// @TEST-ASSERT
AssertTrue(Condition := equal, Message := 'Did not convert LREAL to DINT correctly');
AssertTrue(Condition := converted, Message := 'Did not report LREAL to DINT conversion was successful');

TEST_FINISHED();
END_METHOD

METHOD PUBLIC Check_LREAL_TO_DT_Min
VAR
	value : LREAL := DatatypeLimits.MIN_VALUE_OF_LREAL_WHICH_CAN_BE_HELD_IN_A_DT;
	actual : DT;
	converted : BOOL;
	equal : BOOL;
END_VAR
TEST('Check_LREAL_TO_DT_Min');

// @TEST-RUN
converted := TryConvert_LREAL_TO_Destination(value, actual);
equal := actual = LREAL_TO_DT(value);

// @TEST-ASSERT
AssertTrue(Condition := equal, Message := 'Did not convert LREAL to DT correctly');
AssertTrue(Condition := converted, Message := 'Did not report LREAL to DT conversion was successful');

TEST_FINISHED();
END_METHOD

METHOD PUBLIC Check_LREAL_TO_DT_TooHigh
VAR
	value : LREAL := DatatypeLimits.LREAL_MAX_VALUE;
	actual : DT;
	converted : BOOL;
END_VAR
TEST('Check_LREAL_TO_DT_TooHigh');

// @TEST-RUN
converted := TryConvert_LREAL_TO_Destination(value, actual);

// @TEST-ASSERT
AssertFalse(Condition := converted, Message := 'Did not report LREAL to DT conversion was prevented');

TEST_FINISHED();
END_METHOD

METHOD PUBLIC Check_LREAL_TO_DT_TooLow
VAR
	value : LREAL := DatatypeLimits.LREAL_MIN_VALUE;
	actual : DT;
	converted : BOOL;
END_VAR
TEST('Check_LREAL_TO_DT_TooLow');

// @TEST-RUN
converted := TryConvert_LREAL_TO_Destination(value, actual);

// @TEST-ASSERT
AssertFalse(Condition := converted, Message := 'Did not report LREAL to DT conversion was prevented');

TEST_FINISHED();
END_METHOD

METHOD PUBLIC Check_LREAL_TO_DT_Max
VAR
	value : LREAL := DatatypeLimits.MAX_VALUE_OF_LREAL_WHICH_CAN_BE_HELD_IN_A_DT;
	actual : DT;
	converted : BOOL;
	equal : BOOL;
END_VAR
TEST('Check_LREAL_TO_DT_Max');

// @TEST-RUN
converted := TryConvert_LREAL_TO_Destination(value, actual);
equal := actual = LREAL_TO_DT(value);

// @TEST-ASSERT
AssertTrue(Condition := equal, Message := 'Did not convert LREAL to DT correctly');
AssertTrue(Condition := converted, Message := 'Did not report LREAL to DT conversion was successful');

TEST_FINISHED();
END_METHOD

METHOD PUBLIC Check_LREAL_TO_DWORD_Min
VAR
	value : LREAL := DatatypeLimits.MIN_VALUE_OF_LREAL_WHICH_CAN_BE_HELD_IN_A_DWORD;
	actual : DWORD;
	converted : BOOL;
	equal : BOOL;
END_VAR
TEST('Check_LREAL_TO_DWORD_Min');

// @TEST-RUN
converted := TryConvert_LREAL_TO_Destination(value, actual);
equal := actual = LREAL_TO_DWORD(value);

// @TEST-ASSERT
AssertTrue(Condition := equal, Message := 'Did not convert LREAL to DWORD correctly');
AssertTrue(Condition := converted, Message := 'Did not report LREAL to DWORD conversion was successful');

TEST_FINISHED();
END_METHOD

METHOD PUBLIC Check_LREAL_TO_DWORD_TooHigh
VAR
	value : LREAL := DatatypeLimits.LREAL_MAX_VALUE;
	actual : DWORD;
	converted : BOOL;
END_VAR
TEST('Check_LREAL_TO_DWORD_TooHigh');

// @TEST-RUN
converted := TryConvert_LREAL_TO_Destination(value, actual);

// @TEST-ASSERT
AssertFalse(Condition := converted, Message := 'Did not report LREAL to DWORD conversion was prevented');

TEST_FINISHED();
END_METHOD

METHOD PUBLIC Check_LREAL_TO_DWORD_TooLow
VAR
	value : LREAL := DatatypeLimits.LREAL_MIN_VALUE;
	actual : DWORD;
	converted : BOOL;
END_VAR
TEST('Check_LREAL_TO_DWORD_TooLow');

// @TEST-RUN
converted := TryConvert_LREAL_TO_Destination(value, actual);

// @TEST-ASSERT
AssertFalse(Condition := converted, Message := 'Did not report LREAL to DWORD conversion was prevented');

TEST_FINISHED();
END_METHOD

METHOD PUBLIC Check_LREAL_TO_DWORD_Max
VAR
	value : LREAL := DatatypeLimits.MAX_VALUE_OF_LREAL_WHICH_CAN_BE_HELD_IN_A_DWORD;
	actual : DWORD;
	converted : BOOL;
	equal : BOOL;
END_VAR
TEST('Check_LREAL_TO_DWORD_Max');

// @TEST-RUN
converted := TryConvert_LREAL_TO_Destination(value, actual);
equal := actual = LREAL_TO_DWORD(value);

// @TEST-ASSERT
AssertTrue(Condition := equal, Message := 'Did not convert LREAL to DWORD correctly');
AssertTrue(Condition := converted, Message := 'Did not report LREAL to DWORD conversion was successful');

TEST_FINISHED();
END_METHOD

METHOD PUBLIC Check_LREAL_TO_INT_Min
VAR
	value : LREAL := DatatypeLimits.MIN_VALUE_OF_LREAL_WHICH_CAN_BE_HELD_IN_A_INT;
	actual : INT;
	converted : BOOL;
	equal : BOOL;
END_VAR
TEST('Check_LREAL_TO_INT_Min');

// @TEST-RUN
converted := TryConvert_LREAL_TO_Destination(value, actual);
equal := actual = LREAL_TO_INT(value);

// @TEST-ASSERT
AssertTrue(Condition := equal, Message := 'Did not convert LREAL to INT correctly');
AssertTrue(Condition := converted, Message := 'Did not report LREAL to INT conversion was successful');

TEST_FINISHED();
END_METHOD

METHOD PUBLIC Check_LREAL_TO_INT_TooHigh
VAR
	value : LREAL := DatatypeLimits.LREAL_MAX_VALUE;
	actual : INT;
	converted : BOOL;
END_VAR
TEST('Check_LREAL_TO_INT_TooHigh');

// @TEST-RUN
converted := TryConvert_LREAL_TO_Destination(value, actual);

// @TEST-ASSERT
AssertFalse(Condition := converted, Message := 'Did not report LREAL to INT conversion was prevented');

TEST_FINISHED();
END_METHOD

METHOD PUBLIC Check_LREAL_TO_INT_TooLow
VAR
	value : LREAL := DatatypeLimits.LREAL_MIN_VALUE;
	actual : INT;
	converted : BOOL;
END_VAR
TEST('Check_LREAL_TO_INT_TooLow');

// @TEST-RUN
converted := TryConvert_LREAL_TO_Destination(value, actual);

// @TEST-ASSERT
AssertFalse(Condition := converted, Message := 'Did not report LREAL to INT conversion was prevented');

TEST_FINISHED();
END_METHOD

METHOD PUBLIC Check_LREAL_TO_INT_Max
VAR
	value : LREAL := DatatypeLimits.MAX_VALUE_OF_LREAL_WHICH_CAN_BE_HELD_IN_A_INT;
	actual : INT;
	converted : BOOL;
	equal : BOOL;
END_VAR
TEST('Check_LREAL_TO_INT_Max');

// @TEST-RUN
converted := TryConvert_LREAL_TO_Destination(value, actual);
equal := actual = LREAL_TO_INT(value);

// @TEST-ASSERT
AssertTrue(Condition := equal, Message := 'Did not convert LREAL to INT correctly');
AssertTrue(Condition := converted, Message := 'Did not report LREAL to INT conversion was successful');

TEST_FINISHED();
END_METHOD

METHOD PUBLIC Check_LREAL_TO_LINT_Min
VAR
	value : LREAL := DatatypeLimits.MIN_VALUE_OF_LREAL_WHICH_CAN_BE_HELD_IN_A_LINT;
	actual : LINT;
	converted : BOOL;
	equal : BOOL;
END_VAR
TEST('Check_LREAL_TO_LINT_Min');

// @TEST-RUN
converted := TryConvert_LREAL_TO_Destination(value, actual);
equal := actual = LREAL_TO_LINT(value);

// @TEST-ASSERT
AssertTrue(Condition := equal, Message := 'Did not convert LREAL to LINT correctly');
AssertTrue(Condition := converted, Message := 'Did not report LREAL to LINT conversion was successful');

TEST_FINISHED();
END_METHOD

METHOD PUBLIC Check_LREAL_TO_LINT_TooHigh
VAR
	value : LREAL := DatatypeLimits.LREAL_MAX_VALUE;
	actual : LINT;
	converted : BOOL;
END_VAR
TEST('Check_LREAL_TO_LINT_TooHigh');

// @TEST-RUN
converted := TryConvert_LREAL_TO_Destination(value, actual);

// @TEST-ASSERT
AssertFalse(Condition := converted, Message := 'Did not report LREAL to LINT conversion was prevented');

TEST_FINISHED();
END_METHOD

METHOD PUBLIC Check_LREAL_TO_LINT_TooLow
VAR
	value : LREAL := DatatypeLimits.LREAL_MIN_VALUE;
	actual : LINT;
	converted : BOOL;
END_VAR
TEST('Check_LREAL_TO_LINT_TooLow');

// @TEST-RUN
converted := TryConvert_LREAL_TO_Destination(value, actual);

// @TEST-ASSERT
AssertFalse(Condition := converted, Message := 'Did not report LREAL to LINT conversion was prevented');

TEST_FINISHED();
END_METHOD

METHOD PUBLIC Check_LREAL_TO_LINT_Max
VAR
	value : LREAL := DatatypeLimits.MAX_VALUE_OF_LREAL_WHICH_CAN_BE_HELD_IN_A_LINT;
	actual : LINT;
	converted : BOOL;
	equal : BOOL;
END_VAR
TEST('Check_LREAL_TO_LINT_Max');

// @TEST-RUN
converted := TryConvert_LREAL_TO_Destination(value, actual);
equal := actual = LREAL_TO_LINT(value);

// @TEST-ASSERT
AssertTrue(Condition := equal, Message := 'Did not convert LREAL to LINT correctly');
AssertTrue(Condition := converted, Message := 'Did not report LREAL to LINT conversion was successful');

TEST_FINISHED();
END_METHOD

METHOD PUBLIC Check_LREAL_TO_LREAL_Min
VAR
	value : LREAL := DatatypeLimits.LREAL_MIN_VALUE;
	actual : LREAL;
	converted : BOOL;
	equal : BOOL;
END_VAR
TEST('Check_LREAL_TO_LREAL_Min');

// @TEST-RUN
converted := TryConvert_LREAL_TO_Destination(value, actual);
equal := actual = value;

// @TEST-ASSERT
AssertTrue(Condition := equal, Message := 'Did not convert LREAL to LREAL correctly');
AssertTrue(Condition := converted, Message := 'Did not report LREAL to LREAL conversion was successful');

TEST_FINISHED();
END_METHOD

METHOD PUBLIC Check_LREAL_TO_LREAL_Max
VAR
	value : LREAL := DatatypeLimits.LREAL_MAX_VALUE;
	actual : LREAL;
	converted : BOOL;
	equal : BOOL;
END_VAR
TEST('Check_LREAL_TO_LREAL_Max');

// @TEST-RUN
converted := TryConvert_LREAL_TO_Destination(value, actual);
equal := actual = value;

// @TEST-ASSERT
AssertTrue(Condition := equal, Message := 'Did not convert LREAL to LREAL correctly');
AssertTrue(Condition := converted, Message := 'Did not report LREAL to LREAL conversion was successful');

TEST_FINISHED();
END_METHOD

METHOD PUBLIC Check_LREAL_TO_LWORD_Min
VAR
	value : LREAL := DatatypeLimits.MIN_VALUE_OF_LREAL_WHICH_CAN_BE_HELD_IN_A_LWORD;
	actual : LWORD;
	converted : BOOL;
	equal : BOOL;
END_VAR
TEST('Check_LREAL_TO_LWORD_Min');

// @TEST-RUN
converted := TryConvert_LREAL_TO_Destination(value, actual);
equal := actual = LREAL_TO_LWORD(value);

// @TEST-ASSERT
AssertTrue(Condition := equal, Message := 'Did not convert LREAL to LWORD correctly');
AssertTrue(Condition := converted, Message := 'Did not report LREAL to LWORD conversion was successful');

TEST_FINISHED();
END_METHOD

METHOD PUBLIC Check_LREAL_TO_LWORD_TooHigh
VAR
	value : LREAL := DatatypeLimits.LREAL_MAX_VALUE;
	actual : LWORD;
	converted : BOOL;
END_VAR
TEST('Check_LREAL_TO_LWORD_TooHigh');

// @TEST-RUN
converted := TryConvert_LREAL_TO_Destination(value, actual);

// @TEST-ASSERT
AssertFalse(Condition := converted, Message := 'Did not report LREAL to LWORD conversion was prevented');

TEST_FINISHED();
END_METHOD

METHOD PUBLIC Check_LREAL_TO_LWORD_TooLow
VAR
	value : LREAL := DatatypeLimits.LREAL_MIN_VALUE;
	actual : LWORD;
	converted : BOOL;
END_VAR
TEST('Check_LREAL_TO_LWORD_TooLow');

// @TEST-RUN
converted := TryConvert_LREAL_TO_Destination(value, actual);

// @TEST-ASSERT
AssertFalse(Condition := converted, Message := 'Did not report LREAL to LWORD conversion was prevented');

TEST_FINISHED();
END_METHOD

METHOD PUBLIC Check_LREAL_TO_LWORD_Max
VAR
	value : LREAL := DatatypeLimits.MAX_VALUE_OF_LREAL_WHICH_CAN_BE_HELD_IN_A_LWORD;
	actual : LWORD;
	converted : BOOL;
	equal : BOOL;
END_VAR
TEST('Check_LREAL_TO_LWORD_Max');

// @TEST-RUN
converted := TryConvert_LREAL_TO_Destination(value, actual);
equal := actual = LREAL_TO_LWORD(value);

// @TEST-ASSERT
AssertTrue(Condition := equal, Message := 'Did not convert LREAL to LWORD correctly');
AssertTrue(Condition := converted, Message := 'Did not report LREAL to LWORD conversion was successful');

TEST_FINISHED();
END_METHOD

METHOD PUBLIC Check_LREAL_TO_REAL_Min
VAR
	value : LREAL := DatatypeLimits.MIN_VALUE_OF_LREAL_WHICH_CAN_BE_HELD_IN_A_REAL;
	actual : REAL;
	converted : BOOL;
	equal : BOOL;
END_VAR
TEST('Check_LREAL_TO_REAL_Min');

// @TEST-RUN
converted := TryConvert_LREAL_TO_Destination(value, actual);
equal := actual = LREAL_TO_REAL(value);

// @TEST-ASSERT
AssertTrue(Condition := equal, Message := 'Did not convert LREAL to REAL correctly');
AssertTrue(Condition := converted, Message := 'Did not report LREAL to REAL conversion was successful');

TEST_FINISHED();
END_METHOD

METHOD PUBLIC Check_LREAL_TO_REAL_TooHigh
VAR
	value : LREAL := DatatypeLimits.LREAL_MAX_VALUE;
	actual : REAL;
	converted : BOOL;
END_VAR
TEST('Check_LREAL_TO_REAL_TooHigh');

// @TEST-RUN
converted := TryConvert_LREAL_TO_Destination(value, actual);

// @TEST-ASSERT
AssertFalse(Condition := converted, Message := 'Did not report LREAL to REAL conversion was prevented');

TEST_FINISHED();
END_METHOD

METHOD PUBLIC Check_LREAL_TO_REAL_TooLow
VAR
	value : LREAL := DatatypeLimits.LREAL_MIN_VALUE;
	actual : REAL;
	converted : BOOL;
END_VAR
TEST('Check_LREAL_TO_REAL_TooLow');

// @TEST-RUN
converted := TryConvert_LREAL_TO_Destination(value, actual);

// @TEST-ASSERT
AssertFalse(Condition := converted, Message := 'Did not report LREAL to REAL conversion was prevented');

TEST_FINISHED();
END_METHOD

METHOD PUBLIC Check_LREAL_TO_REAL_Max
VAR
	value : LREAL := DatatypeLimits.MAX_VALUE_OF_LREAL_WHICH_CAN_BE_HELD_IN_A_REAL;
	actual : REAL;
	converted : BOOL;
	equal : BOOL;
END_VAR
TEST('Check_LREAL_TO_REAL_Max');

// @TEST-RUN
converted := TryConvert_LREAL_TO_Destination(value, actual);
equal := actual = LREAL_TO_REAL(value);

// @TEST-ASSERT
AssertTrue(Condition := equal, Message := 'Did not convert LREAL to REAL correctly');
AssertTrue(Condition := converted, Message := 'Did not report LREAL to REAL conversion was successful');

TEST_FINISHED();
END_METHOD

METHOD PUBLIC Check_LREAL_TO_SINT_Min
VAR
	value : LREAL := DatatypeLimits.MIN_VALUE_OF_LREAL_WHICH_CAN_BE_HELD_IN_A_SINT;
	actual : SINT;
	converted : BOOL;
	equal : BOOL;
END_VAR
TEST('Check_LREAL_TO_SINT_Min');

// @TEST-RUN
converted := TryConvert_LREAL_TO_Destination(value, actual);
equal := actual = LREAL_TO_SINT(value);

// @TEST-ASSERT
AssertTrue(Condition := equal, Message := 'Did not convert LREAL to SINT correctly');
AssertTrue(Condition := converted, Message := 'Did not report LREAL to SINT conversion was successful');

TEST_FINISHED();
END_METHOD

METHOD PUBLIC Check_LREAL_TO_SINT_TooHigh
VAR
	value : LREAL := DatatypeLimits.LREAL_MAX_VALUE;
	actual : SINT;
	converted : BOOL;
END_VAR
TEST('Check_LREAL_TO_SINT_TooHigh');

// @TEST-RUN
converted := TryConvert_LREAL_TO_Destination(value, actual);

// @TEST-ASSERT
AssertFalse(Condition := converted, Message := 'Did not report LREAL to SINT conversion was prevented');

TEST_FINISHED();
END_METHOD

METHOD PUBLIC Check_LREAL_TO_SINT_TooLow
VAR
	value : LREAL := DatatypeLimits.LREAL_MIN_VALUE;
	actual : SINT;
	converted : BOOL;
END_VAR
TEST('Check_LREAL_TO_SINT_TooLow');

// @TEST-RUN
converted := TryConvert_LREAL_TO_Destination(value, actual);

// @TEST-ASSERT
AssertFalse(Condition := converted, Message := 'Did not report LREAL to SINT conversion was prevented');

TEST_FINISHED();
END_METHOD

METHOD PUBLIC Check_LREAL_TO_SINT_Max
VAR
	value : LREAL := DatatypeLimits.MAX_VALUE_OF_LREAL_WHICH_CAN_BE_HELD_IN_A_SINT;
	actual : SINT;
	converted : BOOL;
	equal : BOOL;
END_VAR
TEST('Check_LREAL_TO_SINT_Max');

// @TEST-RUN
converted := TryConvert_LREAL_TO_Destination(value, actual);
equal := actual = LREAL_TO_SINT(value);

// @TEST-ASSERT
AssertTrue(Condition := equal, Message := 'Did not convert LREAL to SINT correctly');
AssertTrue(Condition := converted, Message := 'Did not report LREAL to SINT conversion was successful');

TEST_FINISHED();
END_METHOD

METHOD PUBLIC Check_LREAL_TO_STRING_Min
VAR
	value : LREAL := DatatypeLimits.MIN_VALUE_OF_LREAL_WHICH_CAN_BE_HELD_IN_A_STRING;
	actual : STRING;
	converted : BOOL;
	equal : BOOL;
END_VAR
TEST('Check_LREAL_TO_STRING_Min');

// @TEST-RUN
converted := TryConvert_LREAL_TO_Destination(value, actual);
equal := actual = LREAL_TO_STRING(value);

// @TEST-ASSERT
AssertTrue(Condition := equal, Message := 'Did not convert LREAL to STRING correctly');
AssertTrue(Condition := converted, Message := 'Did not report LREAL to STRING conversion was successful');

TEST_FINISHED();
END_METHOD

METHOD PUBLIC Check_LREAL_TO_STRING_TooHigh
VAR
	value : LREAL := DatatypeLimits.LREAL_MAX_VALUE;
	actual : STRING;
	converted : BOOL;
END_VAR
TEST('Check_LREAL_TO_STRING_TooHigh');

// @TEST-RUN
converted := TryConvert_LREAL_TO_Destination(value, actual);

// @TEST-ASSERT
AssertFalse(Condition := converted, Message := 'Did not report LREAL to STRING conversion was prevented');

TEST_FINISHED();
END_METHOD

METHOD PUBLIC Check_LREAL_TO_STRING_TooLow
VAR
	value : LREAL := DatatypeLimits.LREAL_MIN_VALUE;
	actual : STRING;
	converted : BOOL;
END_VAR
TEST('Check_LREAL_TO_STRING_TooLow');

// @TEST-RUN
converted := TryConvert_LREAL_TO_Destination(value, actual);

// @TEST-ASSERT
AssertFalse(Condition := converted, Message := 'Did not report LREAL to STRING conversion was prevented');

TEST_FINISHED();
END_METHOD

METHOD PUBLIC Check_LREAL_TO_STRING_Max
VAR
	value : LREAL := DatatypeLimits.MAX_VALUE_OF_LREAL_WHICH_CAN_BE_HELD_IN_A_STRING;
	actual : STRING;
	converted : BOOL;
	equal : BOOL;
END_VAR
TEST('Check_LREAL_TO_STRING_Max');

// @TEST-RUN
converted := TryConvert_LREAL_TO_Destination(value, actual);
equal := actual = LREAL_TO_STRING(value);

// @TEST-ASSERT
AssertTrue(Condition := equal, Message := 'Did not convert LREAL to STRING correctly');
AssertTrue(Condition := converted, Message := 'Did not report LREAL to STRING conversion was successful');

TEST_FINISHED();
END_METHOD

METHOD PUBLIC Check_LREAL_TO_TIME_Min
VAR
	value : LREAL := DatatypeLimits.MIN_VALUE_OF_LREAL_WHICH_CAN_BE_HELD_IN_A_TIME;
	actual : TIME;
	converted : BOOL;
	equal : BOOL;
END_VAR
TEST('Check_LREAL_TO_TIME_Min');

// @TEST-RUN
converted := TryConvert_LREAL_TO_Destination(value, actual);
equal := actual = LREAL_TO_TIME(value);

// @TEST-ASSERT
AssertTrue(Condition := equal, Message := 'Did not convert LREAL to TIME correctly');
AssertTrue(Condition := converted, Message := 'Did not report LREAL to TIME conversion was successful');

TEST_FINISHED();
END_METHOD

METHOD PUBLIC Check_LREAL_TO_TIME_TooHigh
VAR
	value : LREAL := DatatypeLimits.LREAL_MAX_VALUE;
	actual : TIME;
	converted : BOOL;
END_VAR
TEST('Check_LREAL_TO_TIME_TooHigh');

// @TEST-RUN
converted := TryConvert_LREAL_TO_Destination(value, actual);

// @TEST-ASSERT
AssertFalse(Condition := converted, Message := 'Did not report LREAL to TIME conversion was prevented');

TEST_FINISHED();
END_METHOD

METHOD PUBLIC Check_LREAL_TO_TIME_TooLow
VAR
	value : LREAL := DatatypeLimits.LREAL_MIN_VALUE;
	actual : TIME;
	converted : BOOL;
END_VAR
TEST('Check_LREAL_TO_TIME_TooLow');

// @TEST-RUN
converted := TryConvert_LREAL_TO_Destination(value, actual);

// @TEST-ASSERT
AssertFalse(Condition := converted, Message := 'Did not report LREAL to TIME conversion was prevented');

TEST_FINISHED();
END_METHOD

METHOD PUBLIC Check_LREAL_TO_TIME_Max
VAR
	value : LREAL := DatatypeLimits.MAX_VALUE_OF_LREAL_WHICH_CAN_BE_HELD_IN_A_TIME;
	actual : TIME;
	converted : BOOL;
	equal : BOOL;
END_VAR
TEST('Check_LREAL_TO_TIME_Max');

// @TEST-RUN
converted := TryConvert_LREAL_TO_Destination(value, actual);
equal := actual = LREAL_TO_TIME(value);

// @TEST-ASSERT
AssertTrue(Condition := equal, Message := 'Did not convert LREAL to TIME correctly');
AssertTrue(Condition := converted, Message := 'Did not report LREAL to TIME conversion was successful');

TEST_FINISHED();
END_METHOD

METHOD PUBLIC Check_LREAL_TO_TOD_Min
VAR
	value : LREAL := DatatypeLimits.MIN_VALUE_OF_LREAL_WHICH_CAN_BE_HELD_IN_A_TOD;
	actual : TOD;
	converted : BOOL;
	equal : BOOL;
END_VAR
TEST('Check_LREAL_TO_TOD_Min');

// @TEST-RUN
converted := TryConvert_LREAL_TO_Destination(value, actual);
equal := actual = LREAL_TO_TOD(value);

// @TEST-ASSERT
AssertTrue(Condition := equal, Message := 'Did not convert LREAL to TOD correctly');
AssertTrue(Condition := converted, Message := 'Did not report LREAL to TOD conversion was successful');

TEST_FINISHED();
END_METHOD

METHOD PUBLIC Check_LREAL_TO_TOD_TooHigh
VAR
	value : LREAL := DatatypeLimits.LREAL_MAX_VALUE;
	actual : TOD;
	converted : BOOL;
END_VAR
TEST('Check_LREAL_TO_TOD_TooHigh');

// @TEST-RUN
converted := TryConvert_LREAL_TO_Destination(value, actual);

// @TEST-ASSERT
AssertFalse(Condition := converted, Message := 'Did not report LREAL to TOD conversion was prevented');

TEST_FINISHED();
END_METHOD

METHOD PUBLIC Check_LREAL_TO_TOD_TooLow
VAR
	value : LREAL := DatatypeLimits.LREAL_MIN_VALUE;
	actual : TOD;
	converted : BOOL;
END_VAR
TEST('Check_LREAL_TO_TOD_TooLow');

// @TEST-RUN
converted := TryConvert_LREAL_TO_Destination(value, actual);

// @TEST-ASSERT
AssertFalse(Condition := converted, Message := 'Did not report LREAL to TOD conversion was prevented');

TEST_FINISHED();
END_METHOD

METHOD PUBLIC Check_LREAL_TO_TOD_Max
VAR
	value : LREAL := DatatypeLimits.MAX_VALUE_OF_LREAL_WHICH_CAN_BE_HELD_IN_A_TOD;
	actual : TOD;
	converted : BOOL;
	equal : BOOL;
END_VAR
TEST('Check_LREAL_TO_TOD_Max');

// @TEST-RUN
converted := TryConvert_LREAL_TO_Destination(value, actual);
equal := actual = LREAL_TO_TOD(value);

// @TEST-ASSERT
AssertTrue(Condition := equal, Message := 'Did not convert LREAL to TOD correctly');
AssertTrue(Condition := converted, Message := 'Did not report LREAL to TOD conversion was successful');

TEST_FINISHED();
END_METHOD

METHOD PUBLIC Check_LREAL_TO_UDINT_Min
VAR
	value : LREAL := DatatypeLimits.MIN_VALUE_OF_LREAL_WHICH_CAN_BE_HELD_IN_A_UDINT;
	actual : UDINT;
	converted : BOOL;
	equal : BOOL;
END_VAR
TEST('Check_LREAL_TO_UDINT_Min');

// @TEST-RUN
converted := TryConvert_LREAL_TO_Destination(value, actual);
equal := actual = LREAL_TO_UDINT(value);

// @TEST-ASSERT
AssertTrue(Condition := equal, Message := 'Did not convert LREAL to UDINT correctly');
AssertTrue(Condition := converted, Message := 'Did not report LREAL to UDINT conversion was successful');

TEST_FINISHED();
END_METHOD

METHOD PUBLIC Check_LREAL_TO_UDINT_TooHigh
VAR
	value : LREAL := DatatypeLimits.LREAL_MAX_VALUE;
	actual : UDINT;
	converted : BOOL;
END_VAR
TEST('Check_LREAL_TO_UDINT_TooHigh');

// @TEST-RUN
converted := TryConvert_LREAL_TO_Destination(value, actual);

// @TEST-ASSERT
AssertFalse(Condition := converted, Message := 'Did not report LREAL to UDINT conversion was prevented');

TEST_FINISHED();
END_METHOD

METHOD PUBLIC Check_LREAL_TO_UDINT_TooLow
VAR
	value : LREAL := DatatypeLimits.LREAL_MIN_VALUE;
	actual : UDINT;
	converted : BOOL;
END_VAR
TEST('Check_LREAL_TO_UDINT_TooLow');

// @TEST-RUN
converted := TryConvert_LREAL_TO_Destination(value, actual);

// @TEST-ASSERT
AssertFalse(Condition := converted, Message := 'Did not report LREAL to UDINT conversion was prevented');

TEST_FINISHED();
END_METHOD

METHOD PUBLIC Check_LREAL_TO_UDINT_Max
VAR
	value : LREAL := DatatypeLimits.MAX_VALUE_OF_LREAL_WHICH_CAN_BE_HELD_IN_A_UDINT;
	actual : UDINT;
	converted : BOOL;
	equal : BOOL;
END_VAR
TEST('Check_LREAL_TO_UDINT_Max');

// @TEST-RUN
converted := TryConvert_LREAL_TO_Destination(value, actual);
equal := actual = LREAL_TO_UDINT(value);

// @TEST-ASSERT
AssertTrue(Condition := equal, Message := 'Did not convert LREAL to UDINT correctly');
AssertTrue(Condition := converted, Message := 'Did not report LREAL to UDINT conversion was successful');

TEST_FINISHED();
END_METHOD

METHOD PUBLIC Check_LREAL_TO_UINT_Min
VAR
	value : LREAL := DatatypeLimits.MIN_VALUE_OF_LREAL_WHICH_CAN_BE_HELD_IN_A_UINT;
	actual : UINT;
	converted : BOOL;
	equal : BOOL;
END_VAR
TEST('Check_LREAL_TO_UINT_Min');

// @TEST-RUN
converted := TryConvert_LREAL_TO_Destination(value, actual);
equal := actual = LREAL_TO_UINT(value);

// @TEST-ASSERT
AssertTrue(Condition := equal, Message := 'Did not convert LREAL to UINT correctly');
AssertTrue(Condition := converted, Message := 'Did not report LREAL to UINT conversion was successful');

TEST_FINISHED();
END_METHOD

METHOD PUBLIC Check_LREAL_TO_UINT_TooHigh
VAR
	value : LREAL := DatatypeLimits.LREAL_MAX_VALUE;
	actual : UINT;
	converted : BOOL;
END_VAR
TEST('Check_LREAL_TO_UINT_TooHigh');

// @TEST-RUN
converted := TryConvert_LREAL_TO_Destination(value, actual);

// @TEST-ASSERT
AssertFalse(Condition := converted, Message := 'Did not report LREAL to UINT conversion was prevented');

TEST_FINISHED();
END_METHOD

METHOD PUBLIC Check_LREAL_TO_UINT_TooLow
VAR
	value : LREAL := DatatypeLimits.LREAL_MIN_VALUE;
	actual : UINT;
	converted : BOOL;
END_VAR
TEST('Check_LREAL_TO_UINT_TooLow');

// @TEST-RUN
converted := TryConvert_LREAL_TO_Destination(value, actual);

// @TEST-ASSERT
AssertFalse(Condition := converted, Message := 'Did not report LREAL to UINT conversion was prevented');

TEST_FINISHED();
END_METHOD

METHOD PUBLIC Check_LREAL_TO_UINT_Max
VAR
	value : LREAL := DatatypeLimits.MAX_VALUE_OF_LREAL_WHICH_CAN_BE_HELD_IN_A_UINT;
	actual : UINT;
	converted : BOOL;
	equal : BOOL;
END_VAR
TEST('Check_LREAL_TO_UINT_Max');

// @TEST-RUN
converted := TryConvert_LREAL_TO_Destination(value, actual);
equal := actual = LREAL_TO_UINT(value);

// @TEST-ASSERT
AssertTrue(Condition := equal, Message := 'Did not convert LREAL to UINT correctly');
AssertTrue(Condition := converted, Message := 'Did not report LREAL to UINT conversion was successful');

TEST_FINISHED();
END_METHOD

METHOD PUBLIC Check_LREAL_TO_ULINT_Min
VAR
	value : LREAL := DatatypeLimits.MIN_VALUE_OF_LREAL_WHICH_CAN_BE_HELD_IN_A_ULINT;
	actual : ULINT;
	converted : BOOL;
	equal : BOOL;
END_VAR
TEST('Check_LREAL_TO_ULINT_Min');

// @TEST-RUN
converted := TryConvert_LREAL_TO_Destination(value, actual);
equal := actual = LREAL_TO_ULINT(value);

// @TEST-ASSERT
AssertTrue(Condition := equal, Message := 'Did not convert LREAL to ULINT correctly');
AssertTrue(Condition := converted, Message := 'Did not report LREAL to ULINT conversion was successful');

TEST_FINISHED();
END_METHOD

METHOD PUBLIC Check_LREAL_TO_ULINT_TooHigh
VAR
	value : LREAL := DatatypeLimits.LREAL_MAX_VALUE;
	actual : ULINT;
	converted : BOOL;
END_VAR
TEST('Check_LREAL_TO_ULINT_TooHigh');

// @TEST-RUN
converted := TryConvert_LREAL_TO_Destination(value, actual);

// @TEST-ASSERT
AssertFalse(Condition := converted, Message := 'Did not report LREAL to ULINT conversion was prevented');

TEST_FINISHED();
END_METHOD

METHOD PUBLIC Check_LREAL_TO_ULINT_TooLow
VAR
	value : LREAL := DatatypeLimits.LREAL_MIN_VALUE;
	actual : ULINT;
	converted : BOOL;
END_VAR
TEST('Check_LREAL_TO_ULINT_TooLow');

// @TEST-RUN
converted := TryConvert_LREAL_TO_Destination(value, actual);

// @TEST-ASSERT
AssertFalse(Condition := converted, Message := 'Did not report LREAL to ULINT conversion was prevented');

TEST_FINISHED();
END_METHOD

METHOD PUBLIC Check_LREAL_TO_ULINT_Max
VAR
	value : LREAL := DatatypeLimits.MAX_VALUE_OF_LREAL_WHICH_CAN_BE_HELD_IN_A_ULINT;
	actual : ULINT;
	converted : BOOL;
	equal : BOOL;
END_VAR
TEST('Check_LREAL_TO_ULINT_Max');

// @TEST-RUN
converted := TryConvert_LREAL_TO_Destination(value, actual);
equal := actual = LREAL_TO_ULINT(value);

// @TEST-ASSERT
AssertTrue(Condition := equal, Message := 'Did not convert LREAL to ULINT correctly');
AssertTrue(Condition := converted, Message := 'Did not report LREAL to ULINT conversion was successful');

TEST_FINISHED();
END_METHOD

METHOD PUBLIC Check_LREAL_TO_USINT_Min
VAR
	value : LREAL := DatatypeLimits.MIN_VALUE_OF_LREAL_WHICH_CAN_BE_HELD_IN_A_USINT;
	actual : USINT;
	converted : BOOL;
	equal : BOOL;
END_VAR
TEST('Check_LREAL_TO_USINT_Min');

// @TEST-RUN
converted := TryConvert_LREAL_TO_Destination(value, actual);
equal := actual = LREAL_TO_USINT(value);

// @TEST-ASSERT
AssertTrue(Condition := equal, Message := 'Did not convert LREAL to USINT correctly');
AssertTrue(Condition := converted, Message := 'Did not report LREAL to USINT conversion was successful');

TEST_FINISHED();
END_METHOD

METHOD PUBLIC Check_LREAL_TO_USINT_TooHigh
VAR
	value : LREAL := DatatypeLimits.LREAL_MAX_VALUE;
	actual : USINT;
	converted : BOOL;
END_VAR
TEST('Check_LREAL_TO_USINT_TooHigh');

// @TEST-RUN
converted := TryConvert_LREAL_TO_Destination(value, actual);

// @TEST-ASSERT
AssertFalse(Condition := converted, Message := 'Did not report LREAL to USINT conversion was prevented');

TEST_FINISHED();
END_METHOD

METHOD PUBLIC Check_LREAL_TO_USINT_TooLow
VAR
	value : LREAL := DatatypeLimits.LREAL_MIN_VALUE;
	actual : USINT;
	converted : BOOL;
END_VAR
TEST('Check_LREAL_TO_USINT_TooLow');

// @TEST-RUN
converted := TryConvert_LREAL_TO_Destination(value, actual);

// @TEST-ASSERT
AssertFalse(Condition := converted, Message := 'Did not report LREAL to USINT conversion was prevented');

TEST_FINISHED();
END_METHOD

METHOD PUBLIC Check_LREAL_TO_USINT_Max
VAR
	value : LREAL := DatatypeLimits.MAX_VALUE_OF_LREAL_WHICH_CAN_BE_HELD_IN_A_USINT;
	actual : USINT;
	converted : BOOL;
	equal : BOOL;
END_VAR
TEST('Check_LREAL_TO_USINT_Max');

// @TEST-RUN
converted := TryConvert_LREAL_TO_Destination(value, actual);
equal := actual = LREAL_TO_USINT(value);

// @TEST-ASSERT
AssertTrue(Condition := equal, Message := 'Did not convert LREAL to USINT correctly');
AssertTrue(Condition := converted, Message := 'Did not report LREAL to USINT conversion was successful');

TEST_FINISHED();
END_METHOD

METHOD PUBLIC Check_LREAL_TO_WORD_Min
VAR
	value : LREAL := DatatypeLimits.MIN_VALUE_OF_LREAL_WHICH_CAN_BE_HELD_IN_A_WORD;
	actual : WORD;
	converted : BOOL;
	equal : BOOL;
END_VAR
TEST('Check_LREAL_TO_WORD_Min');

// @TEST-RUN
converted := TryConvert_LREAL_TO_Destination(value, actual);
equal := actual = LREAL_TO_WORD(value);

// @TEST-ASSERT
AssertTrue(Condition := equal, Message := 'Did not convert LREAL to WORD correctly');
AssertTrue(Condition := converted, Message := 'Did not report LREAL to WORD conversion was successful');

TEST_FINISHED();
END_METHOD

METHOD PUBLIC Check_LREAL_TO_WORD_TooHigh
VAR
	value : LREAL := DatatypeLimits.LREAL_MAX_VALUE;
	actual : WORD;
	converted : BOOL;
END_VAR
TEST('Check_LREAL_TO_WORD_TooHigh');

// @TEST-RUN
converted := TryConvert_LREAL_TO_Destination(value, actual);

// @TEST-ASSERT
AssertFalse(Condition := converted, Message := 'Did not report LREAL to WORD conversion was prevented');

TEST_FINISHED();
END_METHOD

METHOD PUBLIC Check_LREAL_TO_WORD_TooLow
VAR
	value : LREAL := DatatypeLimits.LREAL_MIN_VALUE;
	actual : WORD;
	converted : BOOL;
END_VAR
TEST('Check_LREAL_TO_WORD_TooLow');

// @TEST-RUN
converted := TryConvert_LREAL_TO_Destination(value, actual);

// @TEST-ASSERT
AssertFalse(Condition := converted, Message := 'Did not report LREAL to WORD conversion was prevented');

TEST_FINISHED();
END_METHOD

METHOD PUBLIC Check_LREAL_TO_WORD_Max
VAR
	value : LREAL := DatatypeLimits.MAX_VALUE_OF_LREAL_WHICH_CAN_BE_HELD_IN_A_WORD;
	actual : WORD;
	converted : BOOL;
	equal : BOOL;
END_VAR
TEST('Check_LREAL_TO_WORD_Max');

// @TEST-RUN
converted := TryConvert_LREAL_TO_Destination(value, actual);
equal := actual = LREAL_TO_WORD(value);

// @TEST-ASSERT
AssertTrue(Condition := equal, Message := 'Did not convert LREAL to WORD correctly');
AssertTrue(Condition := converted, Message := 'Did not report LREAL to WORD conversion was successful');

TEST_FINISHED();
END_METHOD

END_FUNCTION_BLOCK

// ---- Tests/TIME_TO_TestSuite.TcPOU
FUNCTION_BLOCK PUBLIC TIME_TO_TestSuite EXTENDS TcUnit.FB_TestSuite
VAR
END_VAR

Check_TIME_TO_BOOL_Max();
Check_TIME_TO_BOOL_Min();
Check_TIME_TO_BYTE_Max();
Check_TIME_TO_BYTE_Min();
Check_TIME_TO_BYTE_TooHigh();
Check_TIME_TO_WORD_Max();
Check_TIME_TO_WORD_Min();
Check_TIME_TO_WORD_TooHigh();
Check_TIME_TO_DWORD_Max();
Check_TIME_TO_DWORD_Min();
Check_TIME_TO_LWORD_Max();
Check_TIME_TO_LWORD_Min();
Check_TIME_TO_SINT_Max();
Check_TIME_TO_SINT_Min();
Check_TIME_TO_SINT_TooHigh();
Check_TIME_TO_INT_Max();
Check_TIME_TO_INT_Min();
Check_TIME_TO_INT_TooHigh();
Check_TIME_TO_DINT_Max();
Check_TIME_TO_DINT_Min();
Check_TIME_TO_DINT_TooHigh();
Check_TIME_TO_LINT_Max();
Check_TIME_TO_LINT_Min();
Check_TIME_TO_USINT_Max();
Check_TIME_TO_USINT_Min();
Check_TIME_TO_USINT_TooHigh();
Check_TIME_TO_UINT_Max();
Check_TIME_TO_UINT_Min();
Check_TIME_TO_UINT_TooHigh();
Check_TIME_TO_UDINT_Max();
Check_TIME_TO_UDINT_Min();
Check_TIME_TO_ULINT_Max();
Check_TIME_TO_ULINT_Min();
Check_TIME_TO_REAL_Max();
Check_TIME_TO_REAL_Min();
Check_TIME_TO_LREAL_Max();
Check_TIME_TO_LREAL_Min();
Check_TIME_TO_TIME_Max();
Check_TIME_TO_TIME_Min();
Check_TIME_TO_TOD_Max();
Check_TIME_TO_TOD_Min();
Check_TIME_TO_TOD_TooHigh();
Check_TIME_TO_DATE_Max();
Check_TIME_TO_DATE_Min();
Check_TIME_TO_DT_Max();
Check_TIME_TO_DT_Min();
Check_TIME_TO_STRING_Max();
Check_TIME_TO_STRING_Min();

METHOD PUBLIC Check_TIME_TO_BOOL_Min
VAR
	value : TIME := DatatypeLimits.TIME_MIN_VALUE;
	actual : BOOL;
	converted : BOOL;
	equal : BOOL;
END_VAR
TEST('Check_TIME_TO_BOOL_Min');

// @TEST-RUN
converted := TryConvert_TIME_TO_Destination(value, actual);
equal := actual = TIME_TO_BOOL(value);

// @TEST-ASSERT
AssertTrue(Condition := equal, Message := 'Did not convert TIME to BOOL correctly');
AssertTrue(Condition := converted, Message := 'Did not report TIME to BOOL conversion was successful');

TEST_FINISHED();
END_METHOD

METHOD PUBLIC Check_TIME_TO_BOOL_Max
VAR
	value : TIME := DatatypeLimits.TIME_MAX_VALUE;
	actual : BOOL;
	converted : BOOL;
	equal : BOOL;
END_VAR
TEST('Check_TIME_TO_BOOL_Max');

// @TEST-RUN
converted := TryConvert_TIME_TO_Destination(value, actual);
equal := actual = TIME_TO_BOOL(value);

// @TEST-ASSERT
AssertTrue(Condition := equal, Message := 'Did not convert TIME to BOOL correctly');
AssertTrue(Condition := converted, Message := 'Did not report TIME to BOOL conversion was successful');

TEST_FINISHED();
END_METHOD

METHOD PUBLIC Check_TIME_TO_BYTE_Min
VAR
	value : TIME := DatatypeLimits.TIME_MIN_VALUE;
	actual : BYTE;
	converted : BOOL;
	equal : BOOL;
END_VAR
TEST('Check_TIME_TO_BYTE_Min');

// @TEST-RUN
converted := TryConvert_TIME_TO_Destination(value, actual);
equal := actual = TIME_TO_BYTE(value);

// @TEST-ASSERT
AssertTrue(Condition := equal, Message := 'Did not convert TIME to BYTE correctly');
AssertTrue(Condition := converted, Message := 'Did not report TIME to BYTE conversion was successful');

TEST_FINISHED();
END_METHOD

METHOD PUBLIC Check_TIME_TO_BYTE_TooHigh
VAR
	value : TIME := DatatypeLimits.TIME_MAX_VALUE;
	actual : BYTE;
	converted : BOOL;
END_VAR
TEST('Check_TIME_TO_BYTE_TooHigh');

// @TEST-RUN
converted := TryConvert_TIME_TO_Destination(value, actual);

// @TEST-ASSERT
AssertFalse(Condition := converted, Message := 'Did not report TIME to BYTE conversion was prevented');

TEST_FINISHED();
END_METHOD

METHOD PUBLIC Check_TIME_TO_BYTE_Max
VAR
	value : TIME := DatatypeLimits.MAX_VALUE_OF_TIME_WHICH_CAN_BE_HELD_IN_A_BYTE;
	actual : BYTE;
	converted : BOOL;
	equal : BOOL;
END_VAR
TEST('Check_TIME_TO_BYTE_Max');

// @TEST-RUN
converted := TryConvert_TIME_TO_Destination(value, actual);
equal := actual = TIME_TO_BYTE(value);

// @TEST-ASSERT
AssertTrue(Condition := equal, Message := 'Did not convert TIME to BYTE correctly');
AssertTrue(Condition := converted, Message := 'Did not report TIME to BYTE conversion was successful');

TEST_FINISHED();
END_METHOD

METHOD PUBLIC Check_TIME_TO_DATE_Min
VAR
	value : TIME := DatatypeLimits.TIME_MIN_VALUE;
	actual : DATE;
	converted : BOOL;
	equal : BOOL;
END_VAR
TEST('Check_TIME_TO_DATE_Min');

// @TEST-RUN
converted := TryConvert_TIME_TO_Destination(value, actual);
equal := actual = TIME_TO_DATE(value);

// @TEST-ASSERT
AssertTrue(Condition := equal, Message := 'Did not convert TIME to DATE correctly');
AssertTrue(Condition := converted, Message := 'Did not report TIME to DATE conversion was successful');

TEST_FINISHED();
END_METHOD

METHOD PUBLIC Check_TIME_TO_DATE_Max
VAR
	value : TIME := DatatypeLimits.TIME_MAX_VALUE;
	actual : DATE;
	converted : BOOL;
	equal : BOOL;
END_VAR
TEST('Check_TIME_TO_DATE_Max');

// @TEST-RUN
converted := TryConvert_TIME_TO_Destination(value, actual);
equal := actual = TIME_TO_DATE(value);

// @TEST-ASSERT
AssertTrue(Condition := equal, Message := 'Did not convert TIME to DATE correctly');
AssertTrue(Condition := converted, Message := 'Did not report TIME to DATE conversion was successful');

TEST_FINISHED();
END_METHOD

METHOD PUBLIC Check_TIME_TO_DINT_Min
VAR
	value : TIME := DatatypeLimits.TIME_MIN_VALUE;
	actual : DINT;
	converted : BOOL;
	equal : BOOL;
END_VAR
TEST('Check_TIME_TO_DINT_Min');

// @TEST-RUN
converted := TryConvert_TIME_TO_Destination(value, actual);
equal := actual = TIME_TO_DINT(value);

// @TEST-ASSERT
AssertTrue(Condition := equal, Message := 'Did not convert TIME to DINT correctly');
AssertTrue(Condition := converted, Message := 'Did not report TIME to DINT conversion was successful');

TEST_FINISHED();
END_METHOD

METHOD PUBLIC Check_TIME_TO_DINT_TooHigh
VAR
	value : TIME := DatatypeLimits.TIME_MAX_VALUE;
	actual : DINT;
	converted : BOOL;
END_VAR
TEST('Check_TIME_TO_DINT_TooHigh');

// @TEST-RUN
converted := TryConvert_TIME_TO_Destination(value, actual);

// @TEST-ASSERT
AssertFalse(Condition := converted, Message := 'Did not report TIME to DINT conversion was prevented');

TEST_FINISHED();
END_METHOD

METHOD PUBLIC Check_TIME_TO_DINT_Max
VAR
	value : TIME := DatatypeLimits.MAX_VALUE_OF_TIME_WHICH_CAN_BE_HELD_IN_A_DINT;
	actual : DINT;
	converted : BOOL;
	equal : BOOL;
END_VAR
TEST('Check_TIME_TO_DINT_Max');

// @TEST-RUN
converted := TryConvert_TIME_TO_Destination(value, actual);
equal := actual = TIME_TO_DINT(value);

// @TEST-ASSERT
AssertTrue(Condition := equal, Message := 'Did not convert TIME to DINT correctly');
AssertTrue(Condition := converted, Message := 'Did not report TIME to DINT conversion was successful');

TEST_FINISHED();
END_METHOD

METHOD PUBLIC Check_TIME_TO_DT_Min
VAR
	value : TIME := DatatypeLimits.TIME_MIN_VALUE;
	actual : DT;
	converted : BOOL;
	equal : BOOL;
END_VAR
TEST('Check_TIME_TO_DT_Min');

// @TEST-RUN
converted := TryConvert_TIME_TO_Destination(value, actual);
equal := actual = TIME_TO_DT(value);

// @TEST-ASSERT
AssertTrue(Condition := equal, Message := 'Did not convert TIME to DT correctly');
AssertTrue(Condition := converted, Message := 'Did not report TIME to DT conversion was successful');

TEST_FINISHED();
END_METHOD

METHOD PUBLIC Check_TIME_TO_DT_Max
VAR
	value : TIME := DatatypeLimits.TIME_MAX_VALUE;
	actual : DT;
	converted : BOOL;
	equal : BOOL;
END_VAR
TEST('Check_TIME_TO_DT_Max');

// @TEST-RUN
converted := TryConvert_TIME_TO_Destination(value, actual);
equal := actual = TIME_TO_DT(value);

// @TEST-ASSERT
AssertTrue(Condition := equal, Message := 'Did not convert TIME to DT correctly');
AssertTrue(Condition := converted, Message := 'Did not report TIME to DT conversion was successful');

TEST_FINISHED();
END_METHOD

METHOD PUBLIC Check_TIME_TO_DWORD_Min
VAR
	value : TIME := DatatypeLimits.TIME_MIN_VALUE;
	actual : DWORD;
	converted : BOOL;
	equal : BOOL;
END_VAR
TEST('Check_TIME_TO_DWORD_Min');

// @TEST-RUN
converted := TryConvert_TIME_TO_Destination(value, actual);
equal := actual = TIME_TO_DWORD(value);

// @TEST-ASSERT
AssertTrue(Condition := equal, Message := 'Did not convert TIME to DWORD correctly');
AssertTrue(Condition := converted, Message := 'Did not report TIME to DWORD conversion was successful');

TEST_FINISHED();
END_METHOD

METHOD PUBLIC Check_TIME_TO_DWORD_Max
VAR
	value : TIME := DatatypeLimits.TIME_MAX_VALUE;
	actual : DWORD;
	converted : BOOL;
	equal : BOOL;
END_VAR
TEST('Check_TIME_TO_DWORD_Max');

// @TEST-RUN
converted := TryConvert_TIME_TO_Destination(value, actual);
equal := actual = TIME_TO_DWORD(value);

// @TEST-ASSERT
AssertTrue(Condition := equal, Message := 'Did not convert TIME to DWORD correctly');
AssertTrue(Condition := converted, Message := 'Did not report TIME to DWORD conversion was successful');

TEST_FINISHED();
END_METHOD

METHOD PUBLIC Check_TIME_TO_INT_Min
VAR
	value : TIME := DatatypeLimits.TIME_MIN_VALUE;
	actual : INT;
	converted : BOOL;
	equal : BOOL;
END_VAR
TEST('Check_TIME_TO_INT_Min');

// @TEST-RUN
converted := TryConvert_TIME_TO_Destination(value, actual);
equal := actual = TIME_TO_INT(value);

// @TEST-ASSERT
AssertTrue(Condition := equal, Message := 'Did not convert TIME to INT correctly');
AssertTrue(Condition := converted, Message := 'Did not report TIME to INT conversion was successful');

TEST_FINISHED();
END_METHOD

METHOD PUBLIC Check_TIME_TO_INT_TooHigh
VAR
	value : TIME := DatatypeLimits.TIME_MAX_VALUE;
	actual : INT;
	converted : BOOL;
END_VAR
TEST('Check_TIME_TO_INT_TooHigh');

// @TEST-RUN
converted := TryConvert_TIME_TO_Destination(value, actual);

// @TEST-ASSERT
AssertFalse(Condition := converted, Message := 'Did not report TIME to INT conversion was prevented');

TEST_FINISHED();
END_METHOD

METHOD PUBLIC Check_TIME_TO_INT_Max
VAR
	value : TIME := DatatypeLimits.MAX_VALUE_OF_TIME_WHICH_CAN_BE_HELD_IN_A_INT;
	actual : INT;
	converted : BOOL;
	equal : BOOL;
END_VAR
TEST('Check_TIME_TO_INT_Max');

// @TEST-RUN
converted := TryConvert_TIME_TO_Destination(value, actual);
equal := actual = TIME_TO_INT(value);

// @TEST-ASSERT
AssertTrue(Condition := equal, Message := 'Did not convert TIME to INT correctly');
AssertTrue(Condition := converted, Message := 'Did not report TIME to INT conversion was successful');

TEST_FINISHED();
END_METHOD

METHOD PUBLIC Check_TIME_TO_LINT_Min
VAR
	value : TIME := DatatypeLimits.TIME_MIN_VALUE;
	actual : LINT;
	converted : BOOL;
	equal : BOOL;
END_VAR
TEST('Check_TIME_TO_LINT_Min');

// @TEST-RUN
converted := TryConvert_TIME_TO_Destination(value, actual);
equal := actual = TIME_TO_LINT(value);

// @TEST-ASSERT
AssertTrue(Condition := equal, Message := 'Did not convert TIME to LINT correctly');
AssertTrue(Condition := converted, Message := 'Did not report TIME to LINT conversion was successful');

TEST_FINISHED();
END_METHOD

METHOD PUBLIC Check_TIME_TO_LINT_Max
VAR
	value : TIME := DatatypeLimits.TIME_MAX_VALUE;
	actual : LINT;
	converted : BOOL;
	equal : BOOL;
END_VAR
TEST('Check_TIME_TO_LINT_Max');

// @TEST-RUN
converted := TryConvert_TIME_TO_Destination(value, actual);
equal := actual = TIME_TO_LINT(value);

// @TEST-ASSERT
AssertTrue(Condition := equal, Message := 'Did not convert TIME to LINT correctly');
AssertTrue(Condition := converted, Message := 'Did not report TIME to LINT conversion was successful');

TEST_FINISHED();
END_METHOD

METHOD PUBLIC Check_TIME_TO_LREAL_Min
VAR
	value : TIME := DatatypeLimits.TIME_MIN_VALUE;
	actual : LREAL;
	converted : BOOL;
	equal : BOOL;
END_VAR
TEST('Check_TIME_TO_LREAL_Min');

// @TEST-RUN
converted := TryConvert_TIME_TO_Destination(value, actual);
equal := actual = TIME_TO_LREAL(value);

// @TEST-ASSERT
AssertTrue(Condition := equal, Message := 'Did not convert TIME to LREAL correctly');
AssertTrue(Condition := converted, Message := 'Did not report TIME to LREAL conversion was successful');

TEST_FINISHED();
END_METHOD

METHOD PUBLIC Check_TIME_TO_LREAL_Max
VAR
	value : TIME := DatatypeLimits.TIME_MAX_VALUE;
	actual : LREAL;
	converted : BOOL;
	equal : BOOL;
END_VAR
TEST('Check_TIME_TO_LREAL_Max');

// @TEST-RUN
converted := TryConvert_TIME_TO_Destination(value, actual);
equal := actual = TIME_TO_LREAL(value);

// @TEST-ASSERT
AssertTrue(Condition := equal, Message := 'Did not convert TIME to LREAL correctly');
AssertTrue(Condition := converted, Message := 'Did not report TIME to LREAL conversion was successful');

TEST_FINISHED();
END_METHOD

METHOD PUBLIC Check_TIME_TO_LWORD_Min
VAR
	value : TIME := DatatypeLimits.TIME_MIN_VALUE;
	actual : LWORD;
	converted : BOOL;
	equal : BOOL;
END_VAR
TEST('Check_TIME_TO_LWORD_Min');

// @TEST-RUN
converted := TryConvert_TIME_TO_Destination(value, actual);
equal := actual = TIME_TO_LWORD(value);

// @TEST-ASSERT
AssertTrue(Condition := equal, Message := 'Did not convert TIME to LWORD correctly');
AssertTrue(Condition := converted, Message := 'Did not report TIME to LWORD conversion was successful');

TEST_FINISHED();
END_METHOD

METHOD PUBLIC Check_TIME_TO_LWORD_Max
VAR
	value : TIME := DatatypeLimits.TIME_MAX_VALUE;
	actual : LWORD;
	converted : BOOL;
	equal : BOOL;
END_VAR
TEST('Check_TIME_TO_LWORD_Max');

// @TEST-RUN
converted := TryConvert_TIME_TO_Destination(value, actual);
equal := actual = TIME_TO_LWORD(value);

// @TEST-ASSERT
AssertTrue(Condition := equal, Message := 'Did not convert TIME to LWORD correctly');
AssertTrue(Condition := converted, Message := 'Did not report TIME to LWORD conversion was successful');

TEST_FINISHED();
END_METHOD

METHOD PUBLIC Check_TIME_TO_REAL_Min
VAR
	value : TIME := DatatypeLimits.TIME_MIN_VALUE;
	actual : REAL;
	converted : BOOL;
	equal : BOOL;
END_VAR
TEST('Check_TIME_TO_REAL_Min');

// @TEST-RUN
converted := TryConvert_TIME_TO_Destination(value, actual);
equal := actual = TIME_TO_REAL(value);

// @TEST-ASSERT
AssertTrue(Condition := equal, Message := 'Did not convert TIME to REAL correctly');
AssertTrue(Condition := converted, Message := 'Did not report TIME to REAL conversion was successful');

TEST_FINISHED();
END_METHOD

METHOD PUBLIC Check_TIME_TO_REAL_Max
VAR
	value : TIME := DatatypeLimits.TIME_MAX_VALUE;
	actual : REAL;
	converted : BOOL;
	equal : BOOL;
END_VAR
TEST('Check_TIME_TO_REAL_Max');

// @TEST-RUN
converted := TryConvert_TIME_TO_Destination(value, actual);
equal := actual = TIME_TO_REAL(value);

// @TEST-ASSERT
AssertTrue(Condition := equal, Message := 'Did not convert TIME to REAL correctly');
AssertTrue(Condition := converted, Message := 'Did not report TIME to REAL conversion was successful');

TEST_FINISHED();
END_METHOD

METHOD PUBLIC Check_TIME_TO_SINT_Min
VAR
	value : TIME := DatatypeLimits.TIME_MIN_VALUE;
	actual : SINT;
	converted : BOOL;
	equal : BOOL;
END_VAR
TEST('Check_TIME_TO_SINT_Min');

// @TEST-RUN
converted := TryConvert_TIME_TO_Destination(value, actual);
equal := actual = TIME_TO_SINT(value);

// @TEST-ASSERT
AssertTrue(Condition := equal, Message := 'Did not convert TIME to SINT correctly');
AssertTrue(Condition := converted, Message := 'Did not report TIME to SINT conversion was successful');

TEST_FINISHED();
END_METHOD

METHOD PUBLIC Check_TIME_TO_SINT_TooHigh
VAR
	value : TIME := DatatypeLimits.TIME_MAX_VALUE;
	actual : SINT;
	converted : BOOL;
END_VAR
TEST('Check_TIME_TO_SINT_TooHigh');

// @TEST-RUN
converted := TryConvert_TIME_TO_Destination(value, actual);

// @TEST-ASSERT
AssertFalse(Condition := converted, Message := 'Did not report TIME to SINT conversion was prevented');

TEST_FINISHED();
END_METHOD

METHOD PUBLIC Check_TIME_TO_SINT_Max
VAR
	value : TIME := DatatypeLimits.MAX_VALUE_OF_TIME_WHICH_CAN_BE_HELD_IN_A_SINT;
	actual : SINT;
	converted : BOOL;
	equal : BOOL;
END_VAR
TEST('Check_TIME_TO_SINT_Max');

// @TEST-RUN
converted := TryConvert_TIME_TO_Destination(value, actual);
equal := actual = TIME_TO_SINT(value);

// @TEST-ASSERT
AssertTrue(Condition := equal, Message := 'Did not convert TIME to SINT correctly');
AssertTrue(Condition := converted, Message := 'Did not report TIME to SINT conversion was successful');

TEST_FINISHED();
END_METHOD

METHOD PUBLIC Check_TIME_TO_STRING_Min
VAR
	value : TIME := DatatypeLimits.TIME_MIN_VALUE;
	actual : STRING;
	converted : BOOL;
	equal : BOOL;
END_VAR
TEST('Check_TIME_TO_STRING_Min');

// @TEST-RUN
converted := TryConvert_TIME_TO_Destination(value, actual);
equal := actual = TIME_TO_STRING(value);

// @TEST-ASSERT
AssertTrue(Condition := equal, Message := 'Did not convert TIME to STRING correctly');
AssertTrue(Condition := converted, Message := 'Did not report TIME to STRING conversion was successful');

TEST_FINISHED();
END_METHOD

METHOD PUBLIC Check_TIME_TO_STRING_Max
VAR
	value : TIME := DatatypeLimits.TIME_MAX_VALUE;
	actual : STRING;
	converted : BOOL;
	equal : BOOL;
END_VAR
TEST('Check_TIME_TO_STRING_Max');

// @TEST-RUN
converted := TryConvert_TIME_TO_Destination(value, actual);
equal := actual = TIME_TO_STRING(value);

// @TEST-ASSERT
AssertTrue(Condition := equal, Message := 'Did not convert TIME to STRING correctly');
AssertTrue(Condition := converted, Message := 'Did not report TIME to STRING conversion was successful');

TEST_FINISHED();
END_METHOD

METHOD PUBLIC Check_TIME_TO_TIME_Min
VAR
	value : TIME := DatatypeLimits.TIME_MIN_VALUE;
	actual : TIME;
	converted : BOOL;
	equal : BOOL;
END_VAR
TEST('Check_TIME_TO_TIME_Min');

// @TEST-RUN
converted := TryConvert_TIME_TO_Destination(value, actual);
equal := actual = value;

// @TEST-ASSERT
AssertTrue(Condition := equal, Message := 'Did not convert TIME to TIME correctly');
AssertTrue(Condition := converted, Message := 'Did not report TIME to TIME conversion was successful');

TEST_FINISHED();
END_METHOD

METHOD PUBLIC Check_TIME_TO_TIME_Max
VAR
	value : TIME := DatatypeLimits.TIME_MAX_VALUE;
	actual : TIME;
	converted : BOOL;
	equal : BOOL;
END_VAR
TEST('Check_TIME_TO_TIME_Max');

// @TEST-RUN
converted := TryConvert_TIME_TO_Destination(value, actual);
equal := actual = value;

// @TEST-ASSERT
AssertTrue(Condition := equal, Message := 'Did not convert TIME to TIME correctly');
AssertTrue(Condition := converted, Message := 'Did not report TIME to TIME conversion was successful');

TEST_FINISHED();
END_METHOD

METHOD PUBLIC Check_TIME_TO_TOD_Min
VAR
	value : TIME := DatatypeLimits.TIME_MIN_VALUE;
	actual : TOD;
	converted : BOOL;
	equal : BOOL;
END_VAR
TEST('Check_TIME_TO_TOD_Min');

// @TEST-RUN
converted := TryConvert_TIME_TO_Destination(value, actual);
equal := actual = TIME_TO_TOD(value);

// @TEST-ASSERT
AssertTrue(Condition := equal, Message := 'Did not convert TIME to TOD correctly');
AssertTrue(Condition := converted, Message := 'Did not report TIME to TOD conversion was successful');

TEST_FINISHED();
END_METHOD

METHOD PUBLIC Check_TIME_TO_TOD_TooHigh
VAR
	value : TIME := DatatypeLimits.TIME_MAX_VALUE;
	actual : TOD;
	converted : BOOL;
END_VAR
TEST('Check_TIME_TO_TOD_TooHigh');

// @TEST-RUN
converted := TryConvert_TIME_TO_Destination(value, actual);

// @TEST-ASSERT
AssertFalse(Condition := converted, Message := 'Did not report TIME to TOD conversion was prevented');

TEST_FINISHED();
END_METHOD

METHOD PUBLIC Check_TIME_TO_TOD_Max
VAR
	value : TIME := DatatypeLimits.MAX_VALUE_OF_TIME_WHICH_CAN_BE_HELD_IN_A_TOD;
	actual : TOD;
	converted : BOOL;
	equal : BOOL;
END_VAR
TEST('Check_TIME_TO_TOD_Max');

// @TEST-RUN
converted := TryConvert_TIME_TO_Destination(value, actual);
equal := actual = TIME_TO_TOD(value);

// @TEST-ASSERT
AssertTrue(Condition := equal, Message := 'Did not convert TIME to TOD correctly');
AssertTrue(Condition := converted, Message := 'Did not report TIME to TOD conversion was successful');

TEST_FINISHED();
END_METHOD

METHOD PUBLIC Check_TIME_TO_UDINT_Min
VAR
	value : TIME := DatatypeLimits.TIME_MIN_VALUE;
	actual : UDINT;
	converted : BOOL;
	equal : BOOL;
END_VAR
TEST('Check_TIME_TO_UDINT_Min');

// @TEST-RUN
converted := TryConvert_TIME_TO_Destination(value, actual);
equal := actual = TIME_TO_UDINT(value);

// @TEST-ASSERT
AssertTrue(Condition := equal, Message := 'Did not convert TIME to UDINT correctly');
AssertTrue(Condition := converted, Message := 'Did not report TIME to UDINT conversion was successful');

TEST_FINISHED();
END_METHOD

METHOD PUBLIC Check_TIME_TO_UDINT_Max
VAR
	value : TIME := DatatypeLimits.TIME_MAX_VALUE;
	actual : UDINT;
	converted : BOOL;
	equal : BOOL;
END_VAR
TEST('Check_TIME_TO_UDINT_Max');

// @TEST-RUN
converted := TryConvert_TIME_TO_Destination(value, actual);
equal := actual = TIME_TO_UDINT(value);

// @TEST-ASSERT
AssertTrue(Condition := equal, Message := 'Did not convert TIME to UDINT correctly');
AssertTrue(Condition := converted, Message := 'Did not report TIME to UDINT conversion was successful');

TEST_FINISHED();
END_METHOD

METHOD PUBLIC Check_TIME_TO_UINT_Min
VAR
	value : TIME := DatatypeLimits.TIME_MIN_VALUE;
	actual : UINT;
	converted : BOOL;
	equal : BOOL;
END_VAR
TEST('Check_TIME_TO_UINT_Min');

// @TEST-RUN
converted := TryConvert_TIME_TO_Destination(value, actual);
equal := actual = TIME_TO_UINT(value);

// @TEST-ASSERT
AssertTrue(Condition := equal, Message := 'Did not convert TIME to UINT correctly');
AssertTrue(Condition := converted, Message := 'Did not report TIME to UINT conversion was successful');

TEST_FINISHED();
END_METHOD

METHOD PUBLIC Check_TIME_TO_UINT_TooHigh
VAR
	value : TIME := DatatypeLimits.TIME_MAX_VALUE;
	actual : UINT;
	converted : BOOL;
END_VAR
TEST('Check_TIME_TO_UINT_TooHigh');

// @TEST-RUN
converted := TryConvert_TIME_TO_Destination(value, actual);

// @TEST-ASSERT
AssertFalse(Condition := converted, Message := 'Did not report TIME to UINT conversion was prevented');

TEST_FINISHED();
END_METHOD

METHOD PUBLIC Check_TIME_TO_UINT_Max
VAR
	value : TIME := DatatypeLimits.MAX_VALUE_OF_TIME_WHICH_CAN_BE_HELD_IN_A_UINT;
	actual : UINT;
	converted : BOOL;
	equal : BOOL;
END_VAR
TEST('Check_TIME_TO_UINT_Max');

// @TEST-RUN
converted := TryConvert_TIME_TO_Destination(value, actual);
equal := actual = TIME_TO_UINT(value);

// @TEST-ASSERT
AssertTrue(Condition := equal, Message := 'Did not convert TIME to UINT correctly');
AssertTrue(Condition := converted, Message := 'Did not report TIME to UINT conversion was successful');

TEST_FINISHED();
END_METHOD

METHOD PUBLIC Check_TIME_TO_ULINT_Min
VAR
	value : TIME := DatatypeLimits.TIME_MIN_VALUE;
	actual : ULINT;
	converted : BOOL;
	equal : BOOL;
END_VAR
TEST('Check_TIME_TO_ULINT_Min');

// @TEST-RUN
converted := TryConvert_TIME_TO_Destination(value, actual);
equal := actual = TIME_TO_ULINT(value);

// @TEST-ASSERT
AssertTrue(Condition := equal, Message := 'Did not convert TIME to ULINT correctly');
AssertTrue(Condition := converted, Message := 'Did not report TIME to ULINT conversion was successful');

TEST_FINISHED();
END_METHOD

METHOD PUBLIC Check_TIME_TO_ULINT_Max
VAR
	value : TIME := DatatypeLimits.TIME_MAX_VALUE;
	actual : ULINT;
	converted : BOOL;
	equal : BOOL;
END_VAR
TEST('Check_TIME_TO_ULINT_Max');

// @TEST-RUN
converted := TryConvert_TIME_TO_Destination(value, actual);
equal := actual = TIME_TO_ULINT(value);

// @TEST-ASSERT
AssertTrue(Condition := equal, Message := 'Did not convert TIME to ULINT correctly');
AssertTrue(Condition := converted, Message := 'Did not report TIME to ULINT conversion was successful');

TEST_FINISHED();
END_METHOD

METHOD PUBLIC Check_TIME_TO_USINT_Min
VAR
	value : TIME := DatatypeLimits.TIME_MIN_VALUE;
	actual : USINT;
	converted : BOOL;
	equal : BOOL;
END_VAR
TEST('Check_TIME_TO_USINT_Min');

// @TEST-RUN
converted := TryConvert_TIME_TO_Destination(value, actual);
equal := actual = TIME_TO_USINT(value);

// @TEST-ASSERT
AssertTrue(Condition := equal, Message := 'Did not convert TIME to USINT correctly');
AssertTrue(Condition := converted, Message := 'Did not report TIME to USINT conversion was successful');

TEST_FINISHED();
END_METHOD

METHOD PUBLIC Check_TIME_TO_USINT_TooHigh
VAR
	value : TIME := DatatypeLimits.TIME_MAX_VALUE;
	actual : USINT;
	converted : BOOL;
END_VAR
TEST('Check_TIME_TO_USINT_TooHigh');

// @TEST-RUN
converted := TryConvert_TIME_TO_Destination(value, actual);

// @TEST-ASSERT
AssertFalse(Condition := converted, Message := 'Did not report TIME to USINT conversion was prevented');

TEST_FINISHED();
END_METHOD

METHOD PUBLIC Check_TIME_TO_USINT_Max
VAR
	value : TIME := DatatypeLimits.MAX_VALUE_OF_TIME_WHICH_CAN_BE_HELD_IN_A_USINT;
	actual : USINT;
	converted : BOOL;
	equal : BOOL;
END_VAR
TEST('Check_TIME_TO_USINT_Max');

// @TEST-RUN
converted := TryConvert_TIME_TO_Destination(value, actual);
equal := actual = TIME_TO_USINT(value);

// @TEST-ASSERT
AssertTrue(Condition := equal, Message := 'Did not convert TIME to USINT correctly');
AssertTrue(Condition := converted, Message := 'Did not report TIME to USINT conversion was successful');

TEST_FINISHED();
END_METHOD

METHOD PUBLIC Check_TIME_TO_WORD_Min
VAR
	value : TIME := DatatypeLimits.TIME_MIN_VALUE;
	actual : WORD;
	converted : BOOL;
	equal : BOOL;
END_VAR
TEST('Check_TIME_TO_WORD_Min');

// @TEST-RUN
converted := TryConvert_TIME_TO_Destination(value, actual);
equal := actual = TIME_TO_WORD(value);

// @TEST-ASSERT
AssertTrue(Condition := equal, Message := 'Did not convert TIME to WORD correctly');
AssertTrue(Condition := converted, Message := 'Did not report TIME to WORD conversion was successful');

TEST_FINISHED();
END_METHOD

METHOD PUBLIC Check_TIME_TO_WORD_TooHigh
VAR
	value : TIME := DatatypeLimits.TIME_MAX_VALUE;
	actual : WORD;
	converted : BOOL;
END_VAR
TEST('Check_TIME_TO_WORD_TooHigh');

// @TEST-RUN
converted := TryConvert_TIME_TO_Destination(value, actual);

// @TEST-ASSERT
AssertFalse(Condition := converted, Message := 'Did not report TIME to WORD conversion was prevented');

TEST_FINISHED();
END_METHOD

METHOD PUBLIC Check_TIME_TO_WORD_Max
VAR
	value : TIME := DatatypeLimits.MAX_VALUE_OF_TIME_WHICH_CAN_BE_HELD_IN_A_WORD;
	actual : WORD;
	converted : BOOL;
	equal : BOOL;
END_VAR
TEST('Check_TIME_TO_WORD_Max');

// @TEST-RUN
converted := TryConvert_TIME_TO_Destination(value, actual);
equal := actual = TIME_TO_WORD(value);

// @TEST-ASSERT
AssertTrue(Condition := equal, Message := 'Did not convert TIME to WORD correctly');
AssertTrue(Condition := converted, Message := 'Did not report TIME to WORD conversion was successful');

TEST_FINISHED();
END_METHOD

END_FUNCTION_BLOCK

// ---- Tests/TOD_TO_TestSuite.TcPOU
FUNCTION_BLOCK PUBLIC TOD_TO_TestSuite EXTENDS TcUnit.FB_TestSuite
VAR
END_VAR

Check_TOD_TO_BOOL_Max();
Check_TOD_TO_BOOL_Min();
Check_TOD_TO_BYTE_Max();
Check_TOD_TO_BYTE_Min();
Check_TOD_TO_BYTE_TooHigh();
Check_TOD_TO_WORD_Max();
Check_TOD_TO_WORD_Min();
Check_TOD_TO_WORD_TooHigh();
Check_TOD_TO_DWORD_Max();
Check_TOD_TO_DWORD_Min();
Check_TOD_TO_LWORD_Max();
Check_TOD_TO_LWORD_Min();
Check_TOD_TO_SINT_Max();
Check_TOD_TO_SINT_Min();
Check_TOD_TO_SINT_TooHigh();
Check_TOD_TO_INT_Max();
Check_TOD_TO_INT_Min();
Check_TOD_TO_INT_TooHigh();
Check_TOD_TO_DINT_Max();
Check_TOD_TO_DINT_Min();
Check_TOD_TO_LINT_Max();
Check_TOD_TO_LINT_Min();
Check_TOD_TO_USINT_Max();
Check_TOD_TO_USINT_Min();
Check_TOD_TO_USINT_TooHigh();
Check_TOD_TO_UINT_Max();
Check_TOD_TO_UINT_Min();
Check_TOD_TO_UINT_TooHigh();
Check_TOD_TO_UDINT_Max();
Check_TOD_TO_UDINT_Min();
Check_TOD_TO_ULINT_Max();
Check_TOD_TO_ULINT_Min();
Check_TOD_TO_REAL_Max();
Check_TOD_TO_REAL_Min();
Check_TOD_TO_LREAL_Max();
Check_TOD_TO_LREAL_Min();
Check_TOD_TO_TIME_Max();
Check_TOD_TO_TIME_Min();
Check_TOD_TO_TOD_Max();
Check_TOD_TO_TOD_Min();
Check_TOD_TO_DATE_Max();
Check_TOD_TO_DATE_Min();
Check_TOD_TO_DT_Max();
Check_TOD_TO_DT_Min();
Check_TOD_TO_STRING_Max();
Check_TOD_TO_STRING_Min();

METHOD PUBLIC Check_TOD_TO_BOOL_Min
VAR
	value : TOD := DatatypeLimits.TOD_MIN_VALUE;
	actual : BOOL;
	converted : BOOL;
	equal : BOOL;
END_VAR
TEST('Check_TOD_TO_BOOL_Min');

// @TEST-RUN
converted := TryConvert_TOD_TO_Destination(value, actual);
equal := actual = TOD_TO_BOOL(value);

// @TEST-ASSERT
AssertTrue(Condition := equal, Message := 'Did not convert TOD to BOOL correctly');
AssertTrue(Condition := converted, Message := 'Did not report TOD to BOOL conversion was successful');

TEST_FINISHED();
END_METHOD

METHOD PUBLIC Check_TOD_TO_BOOL_Max
VAR
	value : TOD := DatatypeLimits.TOD_MAX_VALUE;
	actual : BOOL;
	converted : BOOL;
	equal : BOOL;
END_VAR
TEST('Check_TOD_TO_BOOL_Max');

// @TEST-RUN
converted := TryConvert_TOD_TO_Destination(value, actual);
equal := actual = TOD_TO_BOOL(value);

// @TEST-ASSERT
AssertTrue(Condition := equal, Message := 'Did not convert TOD to BOOL correctly');
AssertTrue(Condition := converted, Message := 'Did not report TOD to BOOL conversion was successful');

TEST_FINISHED();
END_METHOD

METHOD PUBLIC Check_TOD_TO_BYTE_Min
VAR
	value : TOD := DatatypeLimits.TOD_MIN_VALUE;
	actual : BYTE;
	converted : BOOL;
	equal : BOOL;
END_VAR
TEST('Check_TOD_TO_BYTE_Min');

// @TEST-RUN
converted := TryConvert_TOD_TO_Destination(value, actual);
equal := actual = TOD_TO_BYTE(value);

// @TEST-ASSERT
AssertTrue(Condition := equal, Message := 'Did not convert TOD to BYTE correctly');
AssertTrue(Condition := converted, Message := 'Did not report TOD to BYTE conversion was successful');

TEST_FINISHED();
END_METHOD

METHOD PUBLIC Check_TOD_TO_BYTE_TooHigh
VAR
	value : TOD := DatatypeLimits.TOD_MAX_VALUE;
	actual : BYTE;
	converted : BOOL;
END_VAR
TEST('Check_TOD_TO_BYTE_TooHigh');

// @TEST-RUN
converted := TryConvert_TOD_TO_Destination(value, actual);

// @TEST-ASSERT
AssertFalse(Condition := converted, Message := 'Did not report TOD to BYTE conversion was prevented');

TEST_FINISHED();
END_METHOD

METHOD PUBLIC Check_TOD_TO_BYTE_Max
VAR
	value : TOD := DatatypeLimits.MAX_VALUE_OF_TOD_WHICH_CAN_BE_HELD_IN_A_BYTE;
	actual : BYTE;
	converted : BOOL;
	equal : BOOL;
END_VAR
TEST('Check_TOD_TO_BYTE_Max');

// @TEST-RUN
converted := TryConvert_TOD_TO_Destination(value, actual);
equal := actual = TOD_TO_BYTE(value);

// @TEST-ASSERT
AssertTrue(Condition := equal, Message := 'Did not convert TOD to BYTE correctly');
AssertTrue(Condition := converted, Message := 'Did not report TOD to BYTE conversion was successful');

TEST_FINISHED();
END_METHOD

METHOD PUBLIC Check_TOD_TO_DATE_Min
VAR
	value : TOD := DatatypeLimits.TOD_MIN_VALUE;
	actual : DATE;
	converted : BOOL;
	equal : BOOL;
END_VAR
TEST('Check_TOD_TO_DATE_Min');

// @TEST-RUN
converted := TryConvert_TOD_TO_Destination(value, actual);
equal := actual = TOD_TO_DATE(value);

// @TEST-ASSERT
AssertTrue(Condition := equal, Message := 'Did not convert TOD to DATE correctly');
AssertTrue(Condition := converted, Message := 'Did not report TOD to DATE conversion was successful');

TEST_FINISHED();
END_METHOD

METHOD PUBLIC Check_TOD_TO_DATE_Max
VAR
	value : TOD := DatatypeLimits.TOD_MAX_VALUE;
	actual : DATE;
	converted : BOOL;
	equal : BOOL;
END_VAR
TEST('Check_TOD_TO_DATE_Max');

// @TEST-RUN
converted := TryConvert_TOD_TO_Destination(value, actual);
equal := actual = TOD_TO_DATE(value);

// @TEST-ASSERT
AssertTrue(Condition := equal, Message := 'Did not convert TOD to DATE correctly');
AssertTrue(Condition := converted, Message := 'Did not report TOD to DATE conversion was successful');

TEST_FINISHED();
END_METHOD

METHOD PUBLIC Check_TOD_TO_DINT_Min
VAR
	value : TOD := DatatypeLimits.TOD_MIN_VALUE;
	actual : DINT;
	converted : BOOL;
	equal : BOOL;
END_VAR
TEST('Check_TOD_TO_DINT_Min');

// @TEST-RUN
converted := TryConvert_TOD_TO_Destination(value, actual);
equal := actual = TOD_TO_DINT(value);

// @TEST-ASSERT
AssertTrue(Condition := equal, Message := 'Did not convert TOD to DINT correctly');
AssertTrue(Condition := converted, Message := 'Did not report TOD to DINT conversion was successful');

TEST_FINISHED();
END_METHOD

METHOD PUBLIC Check_TOD_TO_DINT_Max
VAR
	value : TOD := DatatypeLimits.TOD_MAX_VALUE;
	actual : DINT;
	converted : BOOL;
	equal : BOOL;
END_VAR
TEST('Check_TOD_TO_DINT_Max');

// @TEST-RUN
converted := TryConvert_TOD_TO_Destination(value, actual);
equal := actual = TOD_TO_DINT(value);

// @TEST-ASSERT
AssertTrue(Condition := equal, Message := 'Did not convert TOD to DINT correctly');
AssertTrue(Condition := converted, Message := 'Did not report TOD to DINT conversion was successful');

TEST_FINISHED();
END_METHOD

METHOD PUBLIC Check_TOD_TO_DT_Min
VAR
	value : TOD := DatatypeLimits.TOD_MIN_VALUE;
	actual : DT;
	converted : BOOL;
	equal : BOOL;
END_VAR
TEST('Check_TOD_TO_DT_Min');

// @TEST-RUN
converted := TryConvert_TOD_TO_Destination(value, actual);
equal := actual = TOD_TO_DT(value);

// @TEST-ASSERT
AssertTrue(Condition := equal, Message := 'Did not convert TOD to DT correctly');
AssertTrue(Condition := converted, Message := 'Did not report TOD to DT conversion was successful');

TEST_FINISHED();
END_METHOD

METHOD PUBLIC Check_TOD_TO_DT_Max
VAR
	value : TOD := DatatypeLimits.TOD_MAX_VALUE;
	actual : DT;
	converted : BOOL;
	equal : BOOL;
END_VAR
TEST('Check_TOD_TO_DT_Max');

// @TEST-RUN
converted := TryConvert_TOD_TO_Destination(value, actual);
equal := actual = TOD_TO_DT(value);

// @TEST-ASSERT
AssertTrue(Condition := equal, Message := 'Did not convert TOD to DT correctly');
AssertTrue(Condition := converted, Message := 'Did not report TOD to DT conversion was successful');

TEST_FINISHED();
END_METHOD

METHOD PUBLIC Check_TOD_TO_DWORD_Min
VAR
	value : TOD := DatatypeLimits.TOD_MIN_VALUE;
	actual : DWORD;
	converted : BOOL;
	equal : BOOL;
END_VAR
TEST('Check_TOD_TO_DWORD_Min');

// @TEST-RUN
converted := TryConvert_TOD_TO_Destination(value, actual);
equal := actual = TOD_TO_DWORD(value);

// @TEST-ASSERT
AssertTrue(Condition := equal, Message := 'Did not convert TOD to DWORD correctly');
AssertTrue(Condition := converted, Message := 'Did not report TOD to DWORD conversion was successful');

TEST_FINISHED();
END_METHOD

METHOD PUBLIC Check_TOD_TO_DWORD_Max
VAR
	value : TOD := DatatypeLimits.TOD_MAX_VALUE;
	actual : DWORD;
	converted : BOOL;
	equal : BOOL;
END_VAR
TEST('Check_TOD_TO_DWORD_Max');

// @TEST-RUN
converted := TryConvert_TOD_TO_Destination(value, actual);
equal := actual = TOD_TO_DWORD(value);

// @TEST-ASSERT
AssertTrue(Condition := equal, Message := 'Did not convert TOD to DWORD correctly');
AssertTrue(Condition := converted, Message := 'Did not report TOD to DWORD conversion was successful');

TEST_FINISHED();
END_METHOD

METHOD PUBLIC Check_TOD_TO_INT_Min
VAR
	value : TOD := DatatypeLimits.TOD_MIN_VALUE;
	actual : INT;
	converted : BOOL;
	equal : BOOL;
END_VAR
TEST('Check_TOD_TO_INT_Min');

// @TEST-RUN
converted := TryConvert_TOD_TO_Destination(value, actual);
equal := actual = TOD_TO_INT(value);

// @TEST-ASSERT
AssertTrue(Condition := equal, Message := 'Did not convert TOD to INT correctly');
AssertTrue(Condition := converted, Message := 'Did not report TOD to INT conversion was successful');

TEST_FINISHED();
END_METHOD

METHOD PUBLIC Check_TOD_TO_INT_TooHigh
VAR
	value : TOD := DatatypeLimits.TOD_MAX_VALUE;
	actual : INT;
	converted : BOOL;
END_VAR
TEST('Check_TOD_TO_INT_TooHigh');

// @TEST-RUN
converted := TryConvert_TOD_TO_Destination(value, actual);

// @TEST-ASSERT
AssertFalse(Condition := converted, Message := 'Did not report TOD to INT conversion was prevented');

TEST_FINISHED();
END_METHOD

METHOD PUBLIC Check_TOD_TO_INT_Max
VAR
	value : TOD := DatatypeLimits.MAX_VALUE_OF_TOD_WHICH_CAN_BE_HELD_IN_A_INT;
	actual : INT;
	converted : BOOL;
	equal : BOOL;
END_VAR
TEST('Check_TOD_TO_INT_Max');

// @TEST-RUN
converted := TryConvert_TOD_TO_Destination(value, actual);
equal := actual = TOD_TO_INT(value);

// @TEST-ASSERT
AssertTrue(Condition := equal, Message := 'Did not convert TOD to INT correctly');
AssertTrue(Condition := converted, Message := 'Did not report TOD to INT conversion was successful');

TEST_FINISHED();
END_METHOD

METHOD PUBLIC Check_TOD_TO_LINT_Min
VAR
	value : TOD := DatatypeLimits.TOD_MIN_VALUE;
	actual : LINT;
	converted : BOOL;
	equal : BOOL;
END_VAR
TEST('Check_TOD_TO_LINT_Min');

// @TEST-RUN
converted := TryConvert_TOD_TO_Destination(value, actual);
equal := actual = TOD_TO_LINT(value);

// @TEST-ASSERT
AssertTrue(Condition := equal, Message := 'Did not convert TOD to LINT correctly');
AssertTrue(Condition := converted, Message := 'Did not report TOD to LINT conversion was successful');

TEST_FINISHED();
END_METHOD

METHOD PUBLIC Check_TOD_TO_LINT_Max
VAR
	value : TOD := DatatypeLimits.TOD_MAX_VALUE;
	actual : LINT;
	converted : BOOL;
	equal : BOOL;
END_VAR
TEST('Check_TOD_TO_LINT_Max');

// @TEST-RUN
converted := TryConvert_TOD_TO_Destination(value, actual);
equal := actual = TOD_TO_LINT(value);

// @TEST-ASSERT
AssertTrue(Condition := equal, Message := 'Did not convert TOD to LINT correctly');
AssertTrue(Condition := converted, Message := 'Did not report TOD to LINT conversion was successful');

TEST_FINISHED();
END_METHOD

METHOD PUBLIC Check_TOD_TO_LREAL_Min
VAR
	value : TOD := DatatypeLimits.TOD_MIN_VALUE;
	actual : LREAL;
	converted : BOOL;
	equal : BOOL;
END_VAR
TEST('Check_TOD_TO_LREAL_Min');

// @TEST-RUN
converted := TryConvert_TOD_TO_Destination(value, actual);
equal := actual = TOD_TO_LREAL(value);

// @TEST-ASSERT
AssertTrue(Condition := equal, Message := 'Did not convert TOD to LREAL correctly');
AssertTrue(Condition := converted, Message := 'Did not report TOD to LREAL conversion was successful');

TEST_FINISHED();
END_METHOD

METHOD PUBLIC Check_TOD_TO_LREAL_Max
VAR
	value : TOD := DatatypeLimits.TOD_MAX_VALUE;
	actual : LREAL;
	converted : BOOL;
	equal : BOOL;
END_VAR
TEST('Check_TOD_TO_LREAL_Max');

// @TEST-RUN
converted := TryConvert_TOD_TO_Destination(value, actual);
equal := actual = TOD_TO_LREAL(value);

// @TEST-ASSERT
AssertTrue(Condition := equal, Message := 'Did not convert TOD to LREAL correctly');
AssertTrue(Condition := converted, Message := 'Did not report TOD to LREAL conversion was successful');

TEST_FINISHED();
END_METHOD

METHOD PUBLIC Check_TOD_TO_LWORD_Min
VAR
	value : TOD := DatatypeLimits.TOD_MIN_VALUE;
	actual : LWORD;
	converted : BOOL;
	equal : BOOL;
END_VAR
TEST('Check_TOD_TO_LWORD_Min');

// @TEST-RUN
converted := TryConvert_TOD_TO_Destination(value, actual);
equal := actual = TOD_TO_LWORD(value);

// @TEST-ASSERT
AssertTrue(Condition := equal, Message := 'Did not convert TOD to LWORD correctly');
AssertTrue(Condition := converted, Message := 'Did not report TOD to LWORD conversion was successful');

TEST_FINISHED();
END_METHOD

METHOD PUBLIC Check_TOD_TO_LWORD_Max
VAR
	value : TOD := DatatypeLimits.TOD_MAX_VALUE;
	actual : LWORD;
	converted : BOOL;
	equal : BOOL;
END_VAR
TEST('Check_TOD_TO_LWORD_Max');

// @TEST-RUN
converted := TryConvert_TOD_TO_Destination(value, actual);
equal := actual = TOD_TO_LWORD(value);

// @TEST-ASSERT
AssertTrue(Condition := equal, Message := 'Did not convert TOD to LWORD correctly');
AssertTrue(Condition := converted, Message := 'Did not report TOD to LWORD conversion was successful');

TEST_FINISHED();
END_METHOD

METHOD PUBLIC Check_TOD_TO_REAL_Min
VAR
	value : TOD := DatatypeLimits.TOD_MIN_VALUE;
	actual : REAL;
	converted : BOOL;
	equal : BOOL;
END_VAR
TEST('Check_TOD_TO_REAL_Min');

// @TEST-RUN
converted := TryConvert_TOD_TO_Destination(value, actual);
equal := actual = TOD_TO_REAL(value);

// @TEST-ASSERT
AssertTrue(Condition := equal, Message := 'Did not convert TOD to REAL correctly');
AssertTrue(Condition := converted, Message := 'Did not report TOD to REAL conversion was successful');

TEST_FINISHED();
END_METHOD

METHOD PUBLIC Check_TOD_TO_REAL_Max
VAR
	value : TOD := DatatypeLimits.TOD_MAX_VALUE;
	actual : REAL;
	converted : BOOL;
	equal : BOOL;
END_VAR
TEST('Check_TOD_TO_REAL_Max');

// @TEST-RUN
converted := TryConvert_TOD_TO_Destination(value, actual);
equal := actual = TOD_TO_REAL(value);

// @TEST-ASSERT
AssertTrue(Condition := equal, Message := 'Did not convert TOD to REAL correctly');
AssertTrue(Condition := converted, Message := 'Did not report TOD to REAL conversion was successful');

TEST_FINISHED();
END_METHOD

METHOD PUBLIC Check_TOD_TO_SINT_Min
VAR
	value : TOD := DatatypeLimits.TOD_MIN_VALUE;
	actual : SINT;
	converted : BOOL;
	equal : BOOL;
END_VAR
TEST('Check_TOD_TO_SINT_Min');

// @TEST-RUN
converted := TryConvert_TOD_TO_Destination(value, actual);
equal := actual = TOD_TO_SINT(value);

// @TEST-ASSERT
AssertTrue(Condition := equal, Message := 'Did not convert TOD to SINT correctly');
AssertTrue(Condition := converted, Message := 'Did not report TOD to SINT conversion was successful');

TEST_FINISHED();
END_METHOD

METHOD PUBLIC Check_TOD_TO_SINT_TooHigh
VAR
	value : TOD := DatatypeLimits.TOD_MAX_VALUE;
	actual : SINT;
	converted : BOOL;
END_VAR
TEST('Check_TOD_TO_SINT_TooHigh');

// @TEST-RUN
converted := TryConvert_TOD_TO_Destination(value, actual);

// @TEST-ASSERT
AssertFalse(Condition := converted, Message := 'Did not report TOD to SINT conversion was prevented');

TEST_FINISHED();
END_METHOD

METHOD PUBLIC Check_TOD_TO_SINT_Max
VAR
	value : TOD := DatatypeLimits.MAX_VALUE_OF_TOD_WHICH_CAN_BE_HELD_IN_A_SINT;
	actual : SINT;
	converted : BOOL;
	equal : BOOL;
END_VAR
TEST('Check_TOD_TO_SINT_Max');

// @TEST-RUN
converted := TryConvert_TOD_TO_Destination(value, actual);
equal := actual = TOD_TO_SINT(value);

// @TEST-ASSERT
AssertTrue(Condition := equal, Message := 'Did not convert TOD to SINT correctly');
AssertTrue(Condition := converted, Message := 'Did not report TOD to SINT conversion was successful');

TEST_FINISHED();
END_METHOD

METHOD PUBLIC Check_TOD_TO_STRING_Min
VAR
	value : TOD := DatatypeLimits.TOD_MIN_VALUE;
	actual : STRING;
	converted : BOOL;
	equal : BOOL;
END_VAR
TEST('Check_TOD_TO_STRING_Min');

// @TEST-RUN
converted := TryConvert_TOD_TO_Destination(value, actual);
equal := actual = TOD_TO_STRING(value);

// @TEST-ASSERT
AssertTrue(Condition := equal, Message := 'Did not convert TOD to STRING correctly');
AssertTrue(Condition := converted, Message := 'Did not report TOD to STRING conversion was successful');

TEST_FINISHED();
END_METHOD

METHOD PUBLIC Check_TOD_TO_STRING_Max
VAR
	value : TOD := DatatypeLimits.TOD_MAX_VALUE;
	actual : STRING;
	converted : BOOL;
	equal : BOOL;
END_VAR
TEST('Check_TOD_TO_STRING_Max');

// @TEST-RUN
converted := TryConvert_TOD_TO_Destination(value, actual);
equal := actual = TOD_TO_STRING(value);

// @TEST-ASSERT
AssertTrue(Condition := equal, Message := 'Did not convert TOD to STRING correctly');
AssertTrue(Condition := converted, Message := 'Did not report TOD to STRING conversion was successful');

TEST_FINISHED();
END_METHOD

METHOD PUBLIC Check_TOD_TO_TIME_Min
VAR
	value : TOD := DatatypeLimits.TOD_MIN_VALUE;
	actual : TIME;
	converted : BOOL;
	equal : BOOL;
END_VAR
TEST('Check_TOD_TO_TIME_Min');

// @TEST-RUN
converted := TryConvert_TOD_TO_Destination(value, actual);
equal := actual = TOD_TO_TIME(value);

// @TEST-ASSERT
AssertTrue(Condition := equal, Message := 'Did not convert TOD to TIME correctly');
AssertTrue(Condition := converted, Message := 'Did not report TOD to TIME conversion was successful');

TEST_FINISHED();
END_METHOD

METHOD PUBLIC Check_TOD_TO_TIME_Max
VAR
	value : TOD := DatatypeLimits.TOD_MAX_VALUE;
	actual : TIME;
	converted : BOOL;
	equal : BOOL;
END_VAR
TEST('Check_TOD_TO_TIME_Max');

// @TEST-RUN
converted := TryConvert_TOD_TO_Destination(value, actual);
equal := actual = TOD_TO_TIME(value);

// @TEST-ASSERT
AssertTrue(Condition := equal, Message := 'Did not convert TOD to TIME correctly');
AssertTrue(Condition := converted, Message := 'Did not report TOD to TIME conversion was successful');

TEST_FINISHED();
END_METHOD

METHOD PUBLIC Check_TOD_TO_TOD_Min
VAR
	value : TOD := DatatypeLimits.TOD_MIN_VALUE;
	actual : TOD;
	converted : BOOL;
	equal : BOOL;
END_VAR
TEST('Check_TOD_TO_TOD_Min');

// @TEST-RUN
converted := TryConvert_TOD_TO_Destination(value, actual);
equal := actual = value;

// @TEST-ASSERT
AssertTrue(Condition := equal, Message := 'Did not convert TOD to TOD correctly');
AssertTrue(Condition := converted, Message := 'Did not report TOD to TOD conversion was successful');

TEST_FINISHED();
END_METHOD

METHOD PUBLIC Check_TOD_TO_TOD_Max
VAR
	value : TOD := DatatypeLimits.TOD_MAX_VALUE;
	actual : TOD;
	converted : BOOL;
	equal : BOOL;
END_VAR
TEST('Check_TOD_TO_TOD_Max');

// @TEST-RUN
converted := TryConvert_TOD_TO_Destination(value, actual);
equal := actual = value;

// @TEST-ASSERT
AssertTrue(Condition := equal, Message := 'Did not convert TOD to TOD correctly');
AssertTrue(Condition := converted, Message := 'Did not report TOD to TOD conversion was successful');

TEST_FINISHED();
END_METHOD

METHOD PUBLIC Check_TOD_TO_UDINT_Min
VAR
	value : TOD := DatatypeLimits.TOD_MIN_VALUE;
	actual : UDINT;
	converted : BOOL;
	equal : BOOL;
END_VAR
TEST('Check_TOD_TO_UDINT_Min');

// @TEST-RUN
converted := TryConvert_TOD_TO_Destination(value, actual);
equal := actual = TOD_TO_UDINT(value);

// @TEST-ASSERT
AssertTrue(Condition := equal, Message := 'Did not convert TOD to UDINT correctly');
AssertTrue(Condition := converted, Message := 'Did not report TOD to UDINT conversion was successful');

TEST_FINISHED();
END_METHOD

METHOD PUBLIC Check_TOD_TO_UDINT_Max
VAR
	value : TOD := DatatypeLimits.TOD_MAX_VALUE;
	actual : UDINT;
	converted : BOOL;
	equal : BOOL;
END_VAR
TEST('Check_TOD_TO_UDINT_Max');

// @TEST-RUN
converted := TryConvert_TOD_TO_Destination(value, actual);
equal := actual = TOD_TO_UDINT(value);

// @TEST-ASSERT
AssertTrue(Condition := equal, Message := 'Did not convert TOD to UDINT correctly');
AssertTrue(Condition := converted, Message := 'Did not report TOD to UDINT conversion was successful');

TEST_FINISHED();
END_METHOD

METHOD PUBLIC Check_TOD_TO_UINT_Min
VAR
	value : TOD := DatatypeLimits.TOD_MIN_VALUE;
	actual : UINT;
	converted : BOOL;
	equal : BOOL;
END_VAR
TEST('Check_TOD_TO_UINT_Min');

// @TEST-RUN
converted := TryConvert_TOD_TO_Destination(value, actual);
equal := actual = TOD_TO_UINT(value);

// @TEST-ASSERT
AssertTrue(Condition := equal, Message := 'Did not convert TOD to UINT correctly');
AssertTrue(Condition := converted, Message := 'Did not report TOD to UINT conversion was successful');

TEST_FINISHED();
END_METHOD

METHOD PUBLIC Check_TOD_TO_UINT_TooHigh
VAR
	value : TOD := DatatypeLimits.TOD_MAX_VALUE;
	actual : UINT;
	converted : BOOL;
END_VAR
TEST('Check_TOD_TO_UINT_TooHigh');

// @TEST-RUN
converted := TryConvert_TOD_TO_Destination(value, actual);

// @TEST-ASSERT
AssertFalse(Condition := converted, Message := 'Did not report TOD to UINT conversion was prevented');

TEST_FINISHED();
END_METHOD

METHOD PUBLIC Check_TOD_TO_UINT_Max
VAR
	value : TOD := DatatypeLimits.MAX_VALUE_OF_TOD_WHICH_CAN_BE_HELD_IN_A_UINT;
	actual : UINT;
	converted : BOOL;
	equal : BOOL;
END_VAR
TEST('Check_TOD_TO_UINT_Max');

// @TEST-RUN
converted := TryConvert_TOD_TO_Destination(value, actual);
equal := actual = TOD_TO_UINT(value);

// @TEST-ASSERT
AssertTrue(Condition := equal, Message := 'Did not convert TOD to UINT correctly');
AssertTrue(Condition := converted, Message := 'Did not report TOD to UINT conversion was successful');

TEST_FINISHED();
END_METHOD

METHOD PUBLIC Check_TOD_TO_ULINT_Min
VAR
	value : TOD := DatatypeLimits.TOD_MIN_VALUE;
	actual : ULINT;
	converted : BOOL;
	equal : BOOL;
END_VAR
TEST('Check_TOD_TO_ULINT_Min');

// @TEST-RUN
converted := TryConvert_TOD_TO_Destination(value, actual);
equal := actual = TOD_TO_ULINT(value);

// @TEST-ASSERT
AssertTrue(Condition := equal, Message := 'Did not convert TOD to ULINT correctly');
AssertTrue(Condition := converted, Message := 'Did not report TOD to ULINT conversion was successful');

TEST_FINISHED();
END_METHOD

METHOD PUBLIC Check_TOD_TO_ULINT_Max
VAR
	value : TOD := DatatypeLimits.TOD_MAX_VALUE;
	actual : ULINT;
	converted : BOOL;
	equal : BOOL;
END_VAR
TEST('Check_TOD_TO_ULINT_Max');

// @TEST-RUN
converted := TryConvert_TOD_TO_Destination(value, actual);
equal := actual = TOD_TO_ULINT(value);

// @TEST-ASSERT
AssertTrue(Condition := equal, Message := 'Did not convert TOD to ULINT correctly');
AssertTrue(Condition := converted, Message := 'Did not report TOD to ULINT conversion was successful');

TEST_FINISHED();
END_METHOD

METHOD PUBLIC Check_TOD_TO_USINT_Min
VAR
	value : TOD := DatatypeLimits.TOD_MIN_VALUE;
	actual : USINT;
	converted : BOOL;
	equal : BOOL;
END_VAR
TEST('Check_TOD_TO_USINT_Min');

// @TEST-RUN
converted := TryConvert_TOD_TO_Destination(value, actual);
equal := actual = TOD_TO_USINT(value);

// @TEST-ASSERT
AssertTrue(Condition := equal, Message := 'Did not convert TOD to USINT correctly');
AssertTrue(Condition := converted, Message := 'Did not report TOD to USINT conversion was successful');

TEST_FINISHED();
END_METHOD

METHOD PUBLIC Check_TOD_TO_USINT_TooHigh
VAR
	value : TOD := DatatypeLimits.TOD_MAX_VALUE;
	actual : USINT;
	converted : BOOL;
END_VAR
TEST('Check_TOD_TO_USINT_TooHigh');

// @TEST-RUN
converted := TryConvert_TOD_TO_Destination(value, actual);

// @TEST-ASSERT
AssertFalse(Condition := converted, Message := 'Did not report TOD to USINT conversion was prevented');

TEST_FINISHED();
END_METHOD

METHOD PUBLIC Check_TOD_TO_USINT_Max
VAR
	value : TOD := DatatypeLimits.MAX_VALUE_OF_TOD_WHICH_CAN_BE_HELD_IN_A_USINT;
	actual : USINT;
	converted : BOOL;
	equal : BOOL;
END_VAR
TEST('Check_TOD_TO_USINT_Max');

// @TEST-RUN
converted := TryConvert_TOD_TO_Destination(value, actual);
equal := actual = TOD_TO_USINT(value);

// @TEST-ASSERT
AssertTrue(Condition := equal, Message := 'Did not convert TOD to USINT correctly');
AssertTrue(Condition := converted, Message := 'Did not report TOD to USINT conversion was successful');

TEST_FINISHED();
END_METHOD

METHOD PUBLIC Check_TOD_TO_WORD_Min
VAR
	value : TOD := DatatypeLimits.TOD_MIN_VALUE;
	actual : WORD;
	converted : BOOL;
	equal : BOOL;
END_VAR
TEST('Check_TOD_TO_WORD_Min');

// @TEST-RUN
converted := TryConvert_TOD_TO_Destination(value, actual);
equal := actual = TOD_TO_WORD(value);

// @TEST-ASSERT
AssertTrue(Condition := equal, Message := 'Did not convert TOD to WORD correctly');
AssertTrue(Condition := converted, Message := 'Did not report TOD to WORD conversion was successful');

TEST_FINISHED();
END_METHOD

METHOD PUBLIC Check_TOD_TO_WORD_TooHigh
VAR
	value : TOD := DatatypeLimits.TOD_MAX_VALUE;
	actual : WORD;
	converted : BOOL;
END_VAR
TEST('Check_TOD_TO_WORD_TooHigh');

// @TEST-RUN
converted := TryConvert_TOD_TO_Destination(value, actual);

// @TEST-ASSERT
AssertFalse(Condition := converted, Message := 'Did not report TOD to WORD conversion was prevented');

TEST_FINISHED();
END_METHOD

METHOD PUBLIC Check_TOD_TO_WORD_Max
VAR
	value : TOD := DatatypeLimits.MAX_VALUE_OF_TOD_WHICH_CAN_BE_HELD_IN_A_WORD;
	actual : WORD;
	converted : BOOL;
	equal : BOOL;
END_VAR
TEST('Check_TOD_TO_WORD_Max');

// @TEST-RUN
converted := TryConvert_TOD_TO_Destination(value, actual);
equal := actual = TOD_TO_WORD(value);

// @TEST-ASSERT
AssertTrue(Condition := equal, Message := 'Did not convert TOD to WORD correctly');
AssertTrue(Condition := converted, Message := 'Did not report TOD to WORD conversion was successful');

TEST_FINISHED();
END_METHOD

END_FUNCTION_BLOCK

// ---- Tests/DATE_TO_TestSuite.TcPOU
FUNCTION_BLOCK PUBLIC DATE_TO_TestSuite EXTENDS TcUnit.FB_TestSuite
VAR
END_VAR

Check_DATE_TO_BOOL_Max();
Check_DATE_TO_BOOL_Min();
Check_DATE_TO_BYTE_Max();
Check_DATE_TO_BYTE_Min();
Check_DATE_TO_BYTE_TooHigh();
Check_DATE_TO_WORD_Max();
Check_DATE_TO_WORD_Min();
Check_DATE_TO_WORD_TooHigh();
Check_DATE_TO_DWORD_Max();
Check_DATE_TO_DWORD_Min();
Check_DATE_TO_LWORD_Max();
Check_DATE_TO_LWORD_Min();
Check_DATE_TO_SINT_Max();
Check_DATE_TO_SINT_Min();
Check_DATE_TO_SINT_TooHigh();
Check_DATE_TO_INT_Max();
Check_DATE_TO_INT_Min();
Check_DATE_TO_INT_TooHigh();
Check_DATE_TO_DINT_Max();
Check_DATE_TO_DINT_Min();
Check_DATE_TO_DINT_TooHigh();
Check_DATE_TO_LINT_Max();
Check_DATE_TO_LINT_Min();
Check_DATE_TO_USINT_Max();
Check_DATE_TO_USINT_Min();
Check_DATE_TO_USINT_TooHigh();
Check_DATE_TO_UINT_Max();
Check_DATE_TO_UINT_Min();
Check_DATE_TO_UINT_TooHigh();
Check_DATE_TO_UDINT_Max();
Check_DATE_TO_UDINT_Min();
Check_DATE_TO_ULINT_Max();
Check_DATE_TO_ULINT_Min();
Check_DATE_TO_REAL_Max();
Check_DATE_TO_REAL_Min();
Check_DATE_TO_LREAL_Max();
Check_DATE_TO_LREAL_Min();
Check_DATE_TO_TIME_Max();
Check_DATE_TO_TIME_Min();
Check_DATE_TO_TIME_TooHigh();
Check_DATE_TO_TOD_Max();
Check_DATE_TO_TOD_Min();
Check_DATE_TO_TOD_TooHigh();
Check_DATE_TO_DATE_Max();
Check_DATE_TO_DATE_Min();
Check_DATE_TO_DT_Max();
Check_DATE_TO_DT_Min();
Check_DATE_TO_STRING_Max();
Check_DATE_TO_STRING_Min();

METHOD PUBLIC Check_DATE_TO_BOOL_Min
VAR
	value : DATE := DatatypeLimits.DATE_MIN_VALUE;
	actual : BOOL;
	converted : BOOL;
	equal : BOOL;
END_VAR
TEST('Check_DATE_TO_BOOL_Min');

// @TEST-RUN
converted := TryConvert_DATE_TO_Destination(value, actual);
equal := actual = DATE_TO_BOOL(value);

// @TEST-ASSERT
AssertTrue(Condition := equal, Message := 'Did not convert DATE to BOOL correctly');
AssertTrue(Condition := converted, Message := 'Did not report DATE to BOOL conversion was successful');

TEST_FINISHED();
END_METHOD

METHOD PUBLIC Check_DATE_TO_BOOL_Max
VAR
	value : DATE := DatatypeLimits.DATE_MAX_VALUE;
	actual : BOOL;
	converted : BOOL;
	equal : BOOL;
END_VAR
TEST('Check_DATE_TO_BOOL_Max');

// @TEST-RUN
converted := TryConvert_DATE_TO_Destination(value, actual);
equal := actual = DATE_TO_BOOL(value);

// @TEST-ASSERT
AssertTrue(Condition := equal, Message := 'Did not convert DATE to BOOL correctly');
AssertTrue(Condition := converted, Message := 'Did not report DATE to BOOL conversion was successful');

TEST_FINISHED();
END_METHOD

METHOD PUBLIC Check_DATE_TO_BYTE_Min
VAR
	value : DATE := DatatypeLimits.DATE_MIN_VALUE;
	actual : BYTE;
	converted : BOOL;
	equal : BOOL;
END_VAR
TEST('Check_DATE_TO_BYTE_Min');

// @TEST-RUN
converted := TryConvert_DATE_TO_Destination(value, actual);
equal := actual = DATE_TO_BYTE(value);

// @TEST-ASSERT
AssertTrue(Condition := equal, Message := 'Did not convert DATE to BYTE correctly');
AssertTrue(Condition := converted, Message := 'Did not report DATE to BYTE conversion was successful');

TEST_FINISHED();
END_METHOD

METHOD PUBLIC Check_DATE_TO_BYTE_TooHigh
VAR
	value : DATE := DatatypeLimits.DATE_MAX_VALUE;
	actual : BYTE;
	converted : BOOL;
END_VAR
TEST('Check_DATE_TO_BYTE_TooHigh');

// @TEST-RUN
converted := TryConvert_DATE_TO_Destination(value, actual);

// @TEST-ASSERT
AssertFalse(Condition := converted, Message := 'Did not report DATE to BYTE conversion was prevented');

TEST_FINISHED();
END_METHOD

METHOD PUBLIC Check_DATE_TO_BYTE_Max
VAR
	value : DATE := DatatypeLimits.MAX_VALUE_OF_DATE_WHICH_CAN_BE_HELD_IN_A_BYTE;
	actual : BYTE;
	converted : BOOL;
	equal : BOOL;
END_VAR
TEST('Check_DATE_TO_BYTE_Max');

// @TEST-RUN
converted := TryConvert_DATE_TO_Destination(value, actual);
equal := actual = DATE_TO_BYTE(value);

// @TEST-ASSERT
AssertTrue(Condition := equal, Message := 'Did not convert DATE to BYTE correctly');
AssertTrue(Condition := converted, Message := 'Did not report DATE to BYTE conversion was successful');

TEST_FINISHED();
END_METHOD

METHOD PUBLIC Check_DATE_TO_DATE_Min
VAR
	value : DATE := DatatypeLimits.DATE_MIN_VALUE;
	actual : DATE;
	converted : BOOL;
	equal : BOOL;
END_VAR
TEST('Check_DATE_TO_DATE_Min');

// @TEST-RUN
converted := TryConvert_DATE_TO_Destination(value, actual);
equal := actual = value;

// @TEST-ASSERT
AssertTrue(Condition := equal, Message := 'Did not convert DATE to DATE correctly');
AssertTrue(Condition := converted, Message := 'Did not report DATE to DATE conversion was successful');

TEST_FINISHED();
END_METHOD

METHOD PUBLIC Check_DATE_TO_DATE_Max
VAR
	value : DATE := DatatypeLimits.DATE_MAX_VALUE;
	actual : DATE;
	converted : BOOL;
	equal : BOOL;
END_VAR
TEST('Check_DATE_TO_DATE_Max');

// @TEST-RUN
converted := TryConvert_DATE_TO_Destination(value, actual);
equal := actual = value;

// @TEST-ASSERT
AssertTrue(Condition := equal, Message := 'Did not convert DATE to DATE correctly');
AssertTrue(Condition := converted, Message := 'Did not report DATE to DATE conversion was successful');

TEST_FINISHED();
END_METHOD

METHOD PUBLIC Check_DATE_TO_DINT_Min
VAR
	value : DATE := DatatypeLimits.DATE_MIN_VALUE;
	actual : DINT;
	converted : BOOL;
	equal : BOOL;
END_VAR
TEST('Check_DATE_TO_DINT_Min');

// @TEST-RUN
converted := TryConvert_DATE_TO_Destination(value, actual);
equal := actual = DATE_TO_DINT(value);

// @TEST-ASSERT
AssertTrue(Condition := equal, Message := 'Did not convert DATE to DINT correctly');
AssertTrue(Condition := converted, Message := 'Did not report DATE to DINT conversion was successful');

TEST_FINISHED();
END_METHOD

METHOD PUBLIC Check_DATE_TO_DINT_TooHigh
VAR
	value : DATE := DatatypeLimits.DATE_MAX_VALUE;
	actual : DINT;
	converted : BOOL;
END_VAR
TEST('Check_DATE_TO_DINT_TooHigh');

// @TEST-RUN
converted := TryConvert_DATE_TO_Destination(value, actual);

// @TEST-ASSERT
AssertFalse(Condition := converted, Message := 'Did not report DATE to DINT conversion was prevented');

TEST_FINISHED();
END_METHOD

METHOD PUBLIC Check_DATE_TO_DINT_Max
VAR
	value : DATE := DatatypeLimits.MAX_VALUE_OF_DATE_WHICH_CAN_BE_HELD_IN_A_DINT;
	actual : DINT;
	converted : BOOL;
	equal : BOOL;
END_VAR
TEST('Check_DATE_TO_DINT_Max');

// @TEST-RUN
converted := TryConvert_DATE_TO_Destination(value, actual);
equal := actual = DATE_TO_DINT(value);

// @TEST-ASSERT
AssertTrue(Condition := equal, Message := 'Did not convert DATE to DINT correctly');
AssertTrue(Condition := converted, Message := 'Did not report DATE to DINT conversion was successful');

TEST_FINISHED();
END_METHOD

METHOD PUBLIC Check_DATE_TO_DT_Min
VAR
	value : DATE := DatatypeLimits.DATE_MIN_VALUE;
	actual : DT;
	converted : BOOL;
	equal : BOOL;
END_VAR
TEST('Check_DATE_TO_DT_Min');

// @TEST-RUN
converted := TryConvert_DATE_TO_Destination(value, actual);
equal := actual = DATE_TO_DT(value);

// @TEST-ASSERT
AssertTrue(Condition := equal, Message := 'Did not convert DATE to DT correctly');
AssertTrue(Condition := converted, Message := 'Did not report DATE to DT conversion was successful');

TEST_FINISHED();
END_METHOD

METHOD PUBLIC Check_DATE_TO_DT_Max
VAR
	value : DATE := DatatypeLimits.MAX_VALUE_OF_DATE_WHICH_CAN_BE_HELD_IN_A_DT;
	actual : DT;
	converted : BOOL;
	equal : BOOL;
END_VAR
TEST('Check_DATE_TO_DT_Max');

// @TEST-RUN
converted := TryConvert_DATE_TO_Destination(value, actual);
equal := actual = DATE_TO_DT(value);

// @TEST-ASSERT
AssertTrue(Condition := equal, Message := 'Did not convert DATE to DT correctly');
AssertTrue(Condition := converted, Message := 'Did not report DATE to DT conversion was successful');

TEST_FINISHED();
END_METHOD

METHOD PUBLIC Check_DATE_TO_DWORD_Min
VAR
	value : DATE := DatatypeLimits.DATE_MIN_VALUE;
	actual : DWORD;
	converted : BOOL;
	equal : BOOL;
END_VAR
TEST('Check_DATE_TO_DWORD_Min');

// @TEST-RUN
converted := TryConvert_DATE_TO_Destination(value, actual);
equal := actual = DATE_TO_DWORD(value);

// @TEST-ASSERT
AssertTrue(Condition := equal, Message := 'Did not convert DATE to DWORD correctly');
AssertTrue(Condition := converted, Message := 'Did not report DATE to DWORD conversion was successful');

TEST_FINISHED();
END_METHOD

METHOD PUBLIC Check_DATE_TO_DWORD_Max
VAR
	value : DATE := DatatypeLimits.DATE_MAX_VALUE;
	actual : DWORD;
	converted : BOOL;
	equal : BOOL;
END_VAR
TEST('Check_DATE_TO_DWORD_Max');

// @TEST-RUN
converted := TryConvert_DATE_TO_Destination(value, actual);
equal := actual = DATE_TO_DWORD(value);

// @TEST-ASSERT
AssertTrue(Condition := equal, Message := 'Did not convert DATE to DWORD correctly');
AssertTrue(Condition := converted, Message := 'Did not report DATE to DWORD conversion was successful');

TEST_FINISHED();
END_METHOD

METHOD PUBLIC Check_DATE_TO_INT_Min
VAR
	value : DATE := DatatypeLimits.DATE_MIN_VALUE;
	actual : INT;
	converted : BOOL;
	equal : BOOL;
END_VAR
TEST('Check_DATE_TO_INT_Min');

// @TEST-RUN
converted := TryConvert_DATE_TO_Destination(value, actual);
equal := actual = DATE_TO_INT(value);

// @TEST-ASSERT
AssertTrue(Condition := equal, Message := 'Did not convert DATE to INT correctly');
AssertTrue(Condition := converted, Message := 'Did not report DATE to INT conversion was successful');

TEST_FINISHED();
END_METHOD

METHOD PUBLIC Check_DATE_TO_INT_TooHigh
VAR
	value : DATE := DatatypeLimits.DATE_MAX_VALUE;
	actual : INT;
	converted : BOOL;
END_VAR
TEST('Check_DATE_TO_INT_TooHigh');

// @TEST-RUN
converted := TryConvert_DATE_TO_Destination(value, actual);

// @TEST-ASSERT
AssertFalse(Condition := converted, Message := 'Did not report DATE to INT conversion was prevented');

TEST_FINISHED();
END_METHOD

METHOD PUBLIC Check_DATE_TO_INT_Max
VAR
	value : DATE := DatatypeLimits.MAX_VALUE_OF_DATE_WHICH_CAN_BE_HELD_IN_A_INT;
	actual : INT;
	converted : BOOL;
	equal : BOOL;
END_VAR
TEST('Check_DATE_TO_INT_Max');

// @TEST-RUN
converted := TryConvert_DATE_TO_Destination(value, actual);
equal := actual = DATE_TO_INT(value);

// @TEST-ASSERT
AssertTrue(Condition := equal, Message := 'Did not convert DATE to INT correctly');
AssertTrue(Condition := converted, Message := 'Did not report DATE to INT conversion was successful');

TEST_FINISHED();
END_METHOD

METHOD PUBLIC Check_DATE_TO_LINT_Min
VAR
	value : DATE := DatatypeLimits.DATE_MIN_VALUE;
	actual : LINT;
	converted : BOOL;
	equal : BOOL;
END_VAR
TEST('Check_DATE_TO_LINT_Min');

// @TEST-RUN
converted := TryConvert_DATE_TO_Destination(value, actual);
equal := actual = DATE_TO_LINT(value);

// @TEST-ASSERT
AssertTrue(Condition := equal, Message := 'Did not convert DATE to LINT correctly');
AssertTrue(Condition := converted, Message := 'Did not report DATE to LINT conversion was successful');

TEST_FINISHED();
END_METHOD

METHOD PUBLIC Check_DATE_TO_LINT_Max
VAR
	value : DATE := DatatypeLimits.DATE_MAX_VALUE;
	actual : LINT;
	converted : BOOL;
	equal : BOOL;
END_VAR
TEST('Check_DATE_TO_LINT_Max');

// @TEST-RUN
converted := TryConvert_DATE_TO_Destination(value, actual);
equal := actual = DATE_TO_LINT(value);

// @TEST-ASSERT
AssertTrue(Condition := equal, Message := 'Did not convert DATE to LINT correctly');
AssertTrue(Condition := converted, Message := 'Did not report DATE to LINT conversion was successful');

TEST_FINISHED();
END_METHOD

METHOD PUBLIC Check_DATE_TO_LREAL_Min
VAR
	value : DATE := DatatypeLimits.DATE_MIN_VALUE;
	actual : LREAL;
	converted : BOOL;
	equal : BOOL;
END_VAR
TEST('Check_DATE_TO_LREAL_Min');

// @TEST-RUN
converted := TryConvert_DATE_TO_Destination(value, actual);
equal := actual = DATE_TO_LREAL(value);

// @TEST-ASSERT
AssertTrue(Condition := equal, Message := 'Did not convert DATE to LREAL correctly');
AssertTrue(Condition := converted, Message := 'Did not report DATE to LREAL conversion was successful');

TEST_FINISHED();
END_METHOD

METHOD PUBLIC Check_DATE_TO_LREAL_Max
VAR
	value : DATE := DatatypeLimits.DATE_MAX_VALUE;
	actual : LREAL;
	converted : BOOL;
	equal : BOOL;
END_VAR
TEST('Check_DATE_TO_LREAL_Max');

// @TEST-RUN
converted := TryConvert_DATE_TO_Destination(value, actual);
equal := actual = DATE_TO_LREAL(value);

// @TEST-ASSERT
AssertTrue(Condition := equal, Message := 'Did not convert DATE to LREAL correctly');
AssertTrue(Condition := converted, Message := 'Did not report DATE to LREAL conversion was successful');

TEST_FINISHED();
END_METHOD

METHOD PUBLIC Check_DATE_TO_LWORD_Min
VAR
	value : DATE := DatatypeLimits.DATE_MIN_VALUE;
	actual : LWORD;
	converted : BOOL;
	equal : BOOL;
END_VAR
TEST('Check_DATE_TO_LWORD_Min');

// @TEST-RUN
converted := TryConvert_DATE_TO_Destination(value, actual);
equal := actual = DATE_TO_LWORD(value);

// @TEST-ASSERT
AssertTrue(Condition := equal, Message := 'Did not convert DATE to LWORD correctly');
AssertTrue(Condition := converted, Message := 'Did not report DATE to LWORD conversion was successful');

TEST_FINISHED();
END_METHOD

METHOD PUBLIC Check_DATE_TO_LWORD_Max
VAR
	value : DATE := DatatypeLimits.DATE_MAX_VALUE;
	actual : LWORD;
	converted : BOOL;
	equal : BOOL;
END_VAR
TEST('Check_DATE_TO_LWORD_Max');

// @TEST-RUN
converted := TryConvert_DATE_TO_Destination(value, actual);
equal := actual = DATE_TO_LWORD(value);

// @TEST-ASSERT
AssertTrue(Condition := equal, Message := 'Did not convert DATE to LWORD correctly');
AssertTrue(Condition := converted, Message := 'Did not report DATE to LWORD conversion was successful');

TEST_FINISHED();
END_METHOD

METHOD PUBLIC Check_DATE_TO_REAL_Min
VAR
	value : DATE := DatatypeLimits.DATE_MIN_VALUE;
	actual : REAL;
	converted : BOOL;
	equal : BOOL;
END_VAR
TEST('Check_DATE_TO_REAL_Min');

// @TEST-RUN
converted := TryConvert_DATE_TO_Destination(value, actual);
equal := actual = DATE_TO_REAL(value);

// @TEST-ASSERT
AssertTrue(Condition := equal, Message := 'Did not convert DATE to REAL correctly');
AssertTrue(Condition := converted, Message := 'Did not report DATE to REAL conversion was successful');

TEST_FINISHED();
END_METHOD

METHOD PUBLIC Check_DATE_TO_REAL_Max
VAR
	value : DATE := DatatypeLimits.DATE_MAX_VALUE;
	actual : REAL;
	converted : BOOL;
	equal : BOOL;
END_VAR
TEST('Check_DATE_TO_REAL_Max');

// @TEST-RUN
converted := TryConvert_DATE_TO_Destination(value, actual);
equal := actual = DATE_TO_REAL(value);

// @TEST-ASSERT
AssertTrue(Condition := equal, Message := 'Did not convert DATE to REAL correctly');
AssertTrue(Condition := converted, Message := 'Did not report DATE to REAL conversion was successful');

TEST_FINISHED();
END_METHOD

METHOD PUBLIC Check_DATE_TO_SINT_Min
VAR
	value : DATE := DatatypeLimits.DATE_MIN_VALUE;
	actual : SINT;
	converted : BOOL;
	equal : BOOL;
END_VAR
TEST('Check_DATE_TO_SINT_Min');

// @TEST-RUN
converted := TryConvert_DATE_TO_Destination(value, actual);
equal := actual = DATE_TO_SINT(value);

// @TEST-ASSERT
AssertTrue(Condition := equal, Message := 'Did not convert DATE to SINT correctly');
AssertTrue(Condition := converted, Message := 'Did not report DATE to SINT conversion was successful');

TEST_FINISHED();
END_METHOD

METHOD PUBLIC Check_DATE_TO_SINT_TooHigh
VAR
	value : DATE := DatatypeLimits.DATE_MAX_VALUE;
	actual : SINT;
	converted : BOOL;
END_VAR
TEST('Check_DATE_TO_SINT_TooHigh');

// @TEST-RUN
converted := TryConvert_DATE_TO_Destination(value, actual);

// @TEST-ASSERT
AssertFalse(Condition := converted, Message := 'Did not report DATE to SINT conversion was prevented');

TEST_FINISHED();
END_METHOD

METHOD PUBLIC Check_DATE_TO_SINT_Max
VAR
	value : DATE := DatatypeLimits.MAX_VALUE_OF_DATE_WHICH_CAN_BE_HELD_IN_A_SINT;
	actual : SINT;
	converted : BOOL;
	equal : BOOL;
END_VAR
TEST('Check_DATE_TO_SINT_Max');

// @TEST-RUN
converted := TryConvert_DATE_TO_Destination(value, actual);
equal := actual = DATE_TO_SINT(value);

// @TEST-ASSERT
AssertTrue(Condition := equal, Message := 'Did not convert DATE to SINT correctly');
AssertTrue(Condition := converted, Message := 'Did not report DATE to SINT conversion was successful');

TEST_FINISHED();
END_METHOD

METHOD PUBLIC Check_DATE_TO_STRING_Min
VAR
	value : DATE := DatatypeLimits.DATE_MIN_VALUE;
	actual : STRING;
	converted : BOOL;
	equal : BOOL;
END_VAR
TEST('Check_DATE_TO_STRING_Min');

// @TEST-RUN
converted := TryConvert_DATE_TO_Destination(value, actual);
equal := actual = DATE_TO_STRING(value);

// @TEST-ASSERT
AssertTrue(Condition := equal, Message := 'Did not convert DATE to STRING correctly');
AssertTrue(Condition := converted, Message := 'Did not report DATE to STRING conversion was successful');

TEST_FINISHED();
END_METHOD

METHOD PUBLIC Check_DATE_TO_STRING_Max
VAR
	value : DATE := DatatypeLimits.DATE_MAX_VALUE;
	actual : STRING;
	converted : BOOL;
	equal : BOOL;
END_VAR
TEST('Check_DATE_TO_STRING_Max');

// @TEST-RUN
converted := TryConvert_DATE_TO_Destination(value, actual);
equal := actual = DATE_TO_STRING(value);

// @TEST-ASSERT
AssertTrue(Condition := equal, Message := 'Did not convert DATE to STRING correctly');
AssertTrue(Condition := converted, Message := 'Did not report DATE to STRING conversion was successful');

TEST_FINISHED();
END_METHOD

METHOD PUBLIC Check_DATE_TO_TIME_Min
VAR
	value : DATE := DatatypeLimits.DATE_MIN_VALUE;
	actual : TIME;
	converted : BOOL;
	equal : BOOL;
END_VAR
TEST('Check_DATE_TO_TIME_Min');

// @TEST-RUN
converted := TryConvert_DATE_TO_Destination(value, actual);
equal := actual = DATE_TO_TIME(value);

// @TEST-ASSERT
AssertTrue(Condition := equal, Message := 'Did not convert DATE to TIME correctly');
AssertTrue(Condition := converted, Message := 'Did not report DATE to TIME conversion was successful');

TEST_FINISHED();
END_METHOD

METHOD PUBLIC Check_DATE_TO_TIME_TooHigh
VAR
	value : DATE := DatatypeLimits.DATE_MAX_VALUE;
	actual : TIME;
	converted : BOOL;
END_VAR
TEST('Check_DATE_TO_TIME_TooHigh');

// @TEST-RUN
converted := TryConvert_DATE_TO_Destination(value, actual);

// @TEST-ASSERT
AssertFalse(Condition := converted, Message := 'Did not report DATE to TIME conversion was prevented');

TEST_FINISHED();
END_METHOD

METHOD PUBLIC Check_DATE_TO_TIME_Max
VAR
	value : DATE := DatatypeLimits.MAX_VALUE_OF_DATE_WHICH_CAN_BE_HELD_IN_A_TIME;
	actual : TIME;
	converted : BOOL;
	equal : BOOL;
END_VAR
TEST('Check_DATE_TO_TIME_Max');

// @TEST-RUN
converted := TryConvert_DATE_TO_Destination(value, actual);
equal := actual = DATE_TO_TIME(value);

// @TEST-ASSERT
AssertTrue(Condition := equal, Message := 'Did not convert DATE to TIME correctly');
AssertTrue(Condition := converted, Message := 'Did not report DATE to TIME conversion was successful');

TEST_FINISHED();
END_METHOD

METHOD PUBLIC Check_DATE_TO_TOD_Min
VAR
	value : DATE := DatatypeLimits.DATE_MIN_VALUE;
	actual : TOD;
	converted : BOOL;
	equal : BOOL;
END_VAR
TEST('Check_DATE_TO_TOD_Min');

// @TEST-RUN
converted := TryConvert_DATE_TO_Destination(value, actual);
equal := actual = DATE_TO_TOD(value);

// @TEST-ASSERT
AssertTrue(Condition := equal, Message := 'Did not convert DATE to TOD correctly');
AssertTrue(Condition := converted, Message := 'Did not report DATE to TOD conversion was successful');

